IF SUPER^.Step(882, TRUE, 'Step number 882') THEN
    SUPER^.StepCompleteWhen((_runOneStep OR _runAllSteps) AND _finishStep);

    IF _runOneStep THEN
        _runOneStep := FALSE;
        RETURN;
    END_IF
END_IF

IF SUPER^.Step(883, TRUE, 'Step number 883') THEN
    SUPER^.StepCompleteWhen((_runOneStep OR _runAllSteps) AND _finishStep);

    IF _runOneStep THEN
        _runOneStep := FALSE;
        RETURN;
    END_IF
END_IF

IF SUPER^.Step(884, TRUE, 'Step number 884') THEN
    SUPER^.StepCompleteWhen((_runOneStep OR _runAllSteps) AND _finishStep);

    IF _runOneStep THEN
        _runOneStep := FALSE;
        RETURN;
    END_IF
END_IF

IF SUPER^.Step(885, TRUE, 'Step number 885') THEN
    SUPER^.StepCompleteWhen((_runOneStep OR _runAllSteps) AND _finishStep);

    IF _runOneStep THEN
        _runOneStep := FALSE;
        RETURN;
    END_IF
END_IF

IF SUPER^.Step(886, TRUE, 'Step number 886') THEN
    SUPER^.StepCompleteWhen((_runOneStep OR _runAllSteps) AND _finishStep);

    IF _runOneStep THEN
        _runOneStep := FALSE;
        RETURN;
    END_IF
END_IF

IF SUPER^.Step(887, TRUE, 'Step number 887') THEN
    SUPER^.StepCompleteWhen((_runOneStep OR _runAllSteps) AND _finishStep);

    IF _runOneStep THEN
        _runOneStep := FALSE;
        RETURN;
    END_IF
END_IF

IF SUPER^.Step(888, TRUE, 'Step number 888') THEN
    SUPER^.StepCompleteWhen((_runOneStep OR _runAllSteps) AND _finishStep);

    IF _runOneStep THEN
        _runOneStep := FALSE;
        RETURN;
    END_IF
END_IF

IF SUPER^.Step(889, TRUE, 'Step number 889') THEN
    SUPER^.StepCompleteWhen((_runOneStep OR _runAllSteps) AND _finishStep);

    IF _runOneStep THEN
        _runOneStep := FALSE;
        RETURN;
    END_IF
END_IF

IF SUPER^.Step(890, TRUE, 'Step number 890') THEN
    SUPER^.StepCompleteWhen((_runOneStep OR _runAllSteps) AND _finishStep);

    IF _runOneStep THEN
        _runOneStep := FALSE;
        RETURN;
    END_IF
END_IF

IF SUPER^.Step(891, TRUE, 'Step number 891') THEN
    SUPER^.StepCompleteWhen((_runOneStep OR _runAllSteps) AND _finishStep);

    IF _runOneStep THEN
        _runOneStep := FALSE;
        RETURN;
    END_IF
END_IF

IF SUPER^.Step(892, TRUE, 'Step number 892') THEN
    SUPER^.StepCompleteWhen((_runOneStep OR _runAllSteps) AND _finishStep);

    IF _runOneStep THEN
        _runOneStep := FALSE;
        RETURN;
    END_IF
END_IF

IF SUPER^.Step(893, TRUE, 'Step number 893') THEN
    SUPER^.StepCompleteWhen((_runOneStep OR _runAllSteps) AND _finishStep);

    IF _runOneStep THEN
        _runOneStep := FALSE;
        RETURN;
    END_IF
END_IF

IF SUPER^.Step(894, TRUE, 'Step number 894') THEN
    SUPER^.StepCompleteWhen((_runOneStep OR _runAllSteps) AND _finishStep);

    IF _runOneStep THEN
        _runOneStep := FALSE;
        RETURN;
    END_IF
END_IF

IF SUPER^.Step(895, TRUE, 'Step number 895') THEN
    SUPER^.StepCompleteWhen((_runOneStep OR _runAllSteps) AND _finishStep);

    IF _runOneStep THEN
        _runOneStep := FALSE;
        RETURN;
    END_IF
END_IF

IF SUPER^.Step(896, TRUE, 'Step number 896') THEN
    SUPER^.StepCompleteWhen((_runOneStep OR _runAllSteps) AND _finishStep);

    IF _runOneStep THEN
        _runOneStep := FALSE;
        RETURN;
    END_IF
END_IF

IF SUPER^.Step(897, TRUE, 'Step number 897') THEN
    SUPER^.StepCompleteWhen((_runOneStep OR _runAllSteps) AND _finishStep);

    IF _runOneStep THEN
        _runOneStep := FALSE;
        RETURN;
    END_IF
END_IF

IF SUPER^.Step(898, TRUE, 'Step number 898') THEN
    SUPER^.StepCompleteWhen((_runOneStep OR _runAllSteps) AND _finishStep);

    IF _runOneStep THEN
        _runOneStep := FALSE;
        RETURN;
    END_IF
END_IF

IF SUPER^.Step(899, TRUE, 'Step number 899') THEN
    SUPER^.StepCompleteWhen((_runOneStep OR _runAllSteps) AND _finishStep);

    IF _runOneStep THEN
        _runOneStep := FALSE;
        RETURN;
    END_IF
END_IF

IF SUPER^.Step(900, TRUE, 'Step number 900') THEN
    SUPER^.StepCompleteWhen((_runOneStep OR _runAllSteps) AND _finishStep);

    IF _runOneStep THEN
        _runOneStep := FALSE;
        RETURN;
    END_IF
END_IF

IF SUPER^.Step(901, TRUE, 'Step number 901') THEN
    SUPER^.StepCompleteWhen((_runOneStep OR _runAllSteps) AND _finishStep);

    IF _runOneStep THEN
        _runOneStep := FALSE;
        RETURN;
    END_IF
END_IF

IF SUPER^.Step(902, TRUE, 'Step number 902') THEN
    SUPER^.StepCompleteWhen((_runOneStep OR _runAllSteps) AND _finishStep);

    IF _runOneStep THEN
        _runOneStep := FALSE;
        RETURN;
    END_IF
END_IF

IF SUPER^.Step(903, TRUE, 'Step number 903') THEN
    SUPER^.StepCompleteWhen((_runOneStep OR _runAllSteps) AND _finishStep);

    IF _runOneStep THEN
        _runOneStep := FALSE;
        RETURN;
    END_IF
END_IF

IF SUPER^.Step(904, TRUE, 'Step number 904') THEN
    SUPER^.StepCompleteWhen((_runOneStep OR _runAllSteps) AND _finishStep);

    IF _runOneStep THEN
        _runOneStep := FALSE;
        RETURN;
    END_IF
END_IF

IF SUPER^.Step(905, TRUE, 'Step number 905') THEN
    SUPER^.StepCompleteWhen((_runOneStep OR _runAllSteps) AND _finishStep);

    IF _runOneStep THEN
        _runOneStep := FALSE;
        RETURN;
    END_IF
END_IF

IF SUPER^.Step(906, TRUE, 'Step number 906') THEN
    SUPER^.StepCompleteWhen((_runOneStep OR _runAllSteps) AND _finishStep);

    IF _runOneStep THEN
        _runOneStep := FALSE;
        RETURN;
    END_IF
END_IF

IF SUPER^.Step(907, TRUE, 'Step number 907') THEN
    SUPER^.StepCompleteWhen((_runOneStep OR _runAllSteps) AND _finishStep);

    IF _runOneStep THEN
        _runOneStep := FALSE;
        RETURN;
    END_IF
END_IF

IF SUPER^.Step(908, TRUE, 'Step number 908') THEN
    SUPER^.StepCompleteWhen((_runOneStep OR _runAllSteps) AND _finishStep);

    IF _runOneStep THEN
        _runOneStep := FALSE;
        RETURN;
    END_IF
END_IF

IF SUPER^.Step(909, TRUE, 'Step number 909') THEN
    SUPER^.StepCompleteWhen((_runOneStep OR _runAllSteps) AND _finishStep);

    IF _runOneStep THEN
        _runOneStep := FALSE;
        RETURN;
    END_IF
END_IF

IF SUPER^.Step(910, TRUE, 'Step number 910') THEN
    SUPER^.StepCompleteWhen((_runOneStep OR _runAllSteps) AND _finishStep);

    IF _runOneStep THEN
        _runOneStep := FALSE;
        RETURN;
    END_IF
END_IF

IF SUPER^.Step(911, TRUE, 'Step number 911') THEN
    SUPER^.StepCompleteWhen((_runOneStep OR _runAllSteps) AND _finishStep);

    IF _runOneStep THEN
        _runOneStep := FALSE;
        RETURN;
    END_IF
END_IF

IF SUPER^.Step(912, TRUE, 'Step number 912') THEN
    SUPER^.StepCompleteWhen((_runOneStep OR _runAllSteps) AND _finishStep);

    IF _runOneStep THEN
        _runOneStep := FALSE;
        RETURN;
    END_IF
END_IF

IF SUPER^.Step(913, TRUE, 'Step number 913') THEN
    SUPER^.StepCompleteWhen((_runOneStep OR _runAllSteps) AND _finishStep);

    IF _runOneStep THEN
        _runOneStep := FALSE;
        RETURN;
    END_IF
END_IF

IF SUPER^.Step(914, TRUE, 'Step number 914') THEN
    SUPER^.StepCompleteWhen((_runOneStep OR _runAllSteps) AND _finishStep);

    IF _runOneStep THEN
        _runOneStep := FALSE;
        RETURN;
    END_IF
END_IF

IF SUPER^.Step(915, TRUE, 'Step number 915') THEN
    SUPER^.StepCompleteWhen((_runOneStep OR _runAllSteps) AND _finishStep);

    IF _runOneStep THEN
        _runOneStep := FALSE;
        RETURN;
    END_IF
END_IF

IF SUPER^.Step(916, TRUE, 'Step number 916') THEN
    SUPER^.StepCompleteWhen((_runOneStep OR _runAllSteps) AND _finishStep);

    IF _runOneStep THEN
        _runOneStep := FALSE;
        RETURN;
    END_IF
END_IF

IF SUPER^.Step(917, TRUE, 'Step number 917') THEN
    SUPER^.StepCompleteWhen((_runOneStep OR _runAllSteps) AND _finishStep);

    IF _runOneStep THEN
        _runOneStep := FALSE;
        RETURN;
    END_IF
END_IF

IF SUPER^.Step(918, TRUE, 'Step number 918') THEN
    SUPER^.StepCompleteWhen((_runOneStep OR _runAllSteps) AND _finishStep);

    IF _runOneStep THEN
        _runOneStep := FALSE;
        RETURN;
    END_IF
END_IF

IF SUPER^.Step(919, TRUE, 'Step number 919') THEN
    SUPER^.StepCompleteWhen((_runOneStep OR _runAllSteps) AND _finishStep);

    IF _runOneStep THEN
        _runOneStep := FALSE;
        RETURN;
    END_IF
END_IF

IF SUPER^.Step(920, TRUE, 'Step number 920') THEN
    SUPER^.StepCompleteWhen((_runOneStep OR _runAllSteps) AND _finishStep);

    IF _runOneStep THEN
        _runOneStep := FALSE;
        RETURN;
    END_IF
END_IF

IF SUPER^.Step(921, TRUE, 'Step number 921') THEN
    SUPER^.StepCompleteWhen((_runOneStep OR _runAllSteps) AND _finishStep);

    IF _runOneStep THEN
        _runOneStep := FALSE;
        RETURN;
    END_IF
END_IF

IF SUPER^.Step(922, TRUE, 'Step number 922') THEN
    SUPER^.StepCompleteWhen((_runOneStep OR _runAllSteps) AND _finishStep);

    IF _runOneStep THEN
        _runOneStep := FALSE;
        RETURN;
    END_IF
END_IF

IF SUPER^.Step(923, TRUE, 'Step number 923') THEN
    SUPER^.StepCompleteWhen((_runOneStep OR _runAllSteps) AND _finishStep);

    IF _runOneStep THEN
        _runOneStep := FALSE;
        RETURN;
    END_IF
END_IF

IF SUPER^.Step(924, TRUE, 'Step number 924') THEN
    SUPER^.StepCompleteWhen((_runOneStep OR _runAllSteps) AND _finishStep);

    IF _runOneStep THEN
        _runOneStep := FALSE;
        RETURN;
    END_IF
END_IF

IF SUPER^.Step(925, TRUE, 'Step number 925') THEN
    SUPER^.StepCompleteWhen((_runOneStep OR _runAllSteps) AND _finishStep);

    IF _runOneStep THEN
        _runOneStep := FALSE;
        RETURN;
    END_IF
END_IF

IF SUPER^.Step(926, TRUE, 'Step number 926') THEN
    SUPER^.StepCompleteWhen((_runOneStep OR _runAllSteps) AND _finishStep);

    IF _runOneStep THEN
        _runOneStep := FALSE;
        RETURN;
    END_IF
END_IF

IF SUPER^.Step(927, TRUE, 'Step number 927') THEN
    SUPER^.StepCompleteWhen((_runOneStep OR _runAllSteps) AND _finishStep);

    IF _runOneStep THEN
        _runOneStep := FALSE;
        RETURN;
    END_IF
END_IF

IF SUPER^.Step(928, TRUE, 'Step number 928') THEN
    SUPER^.StepCompleteWhen((_runOneStep OR _runAllSteps) AND _finishStep);

    IF _runOneStep THEN
        _runOneStep := FALSE;
        RETURN;
    END_IF
END_IF

IF SUPER^.Step(929, TRUE, 'Step number 929') THEN
    SUPER^.StepCompleteWhen((_runOneStep OR _runAllSteps) AND _finishStep);

    IF _runOneStep THEN
        _runOneStep := FALSE;
        RETURN;
    END_IF
END_IF

IF SUPER^.Step(930, TRUE, 'Step number 930') THEN
    SUPER^.StepCompleteWhen((_runOneStep OR _runAllSteps) AND _finishStep);

    IF _runOneStep THEN
        _runOneStep := FALSE;
        RETURN;
    END_IF
END_IF

IF SUPER^.Step(931, TRUE, 'Step number 931') THEN
    SUPER^.StepCompleteWhen((_runOneStep OR _runAllSteps) AND _finishStep);

    IF _runOneStep THEN
        _runOneStep := FALSE;
        RETURN;
    END_IF
END_IF

IF SUPER^.Step(932, TRUE, 'Step number 932') THEN
    SUPER^.StepCompleteWhen((_runOneStep OR _runAllSteps) AND _finishStep);

    IF _runOneStep THEN
        _runOneStep := FALSE;
        RETURN;
    END_IF
END_IF

IF SUPER^.Step(933, TRUE, 'Step number 933') THEN
    SUPER^.StepCompleteWhen((_runOneStep OR _runAllSteps) AND _finishStep);

    IF _runOneStep THEN
        _runOneStep := FALSE;
        RETURN;
    END_IF
END_IF

IF SUPER^.Step(934, TRUE, 'Step number 934') THEN
    SUPER^.StepCompleteWhen((_runOneStep OR _runAllSteps) AND _finishStep);

    IF _runOneStep THEN
        _runOneStep := FALSE;
        RETURN;
    END_IF
END_IF

IF SUPER^.Step(935, TRUE, 'Step number 935') THEN
    SUPER^.StepCompleteWhen((_runOneStep OR _runAllSteps) AND _finishStep);

    IF _runOneStep THEN
        _runOneStep := FALSE;
        RETURN;
    END_IF
END_IF

IF SUPER^.Step(936, TRUE, 'Step number 936') THEN
    SUPER^.StepCompleteWhen((_runOneStep OR _runAllSteps) AND _finishStep);

    IF _runOneStep THEN
        _runOneStep := FALSE;
        RETURN;
    END_IF
END_IF

IF SUPER^.Step(937, TRUE, 'Step number 937') THEN
    SUPER^.StepCompleteWhen((_runOneStep OR _runAllSteps) AND _finishStep);

    IF _runOneStep THEN
        _runOneStep := FALSE;
        RETURN;
    END_IF
END_IF

IF SUPER^.Step(938, TRUE, 'Step number 938') THEN
    SUPER^.StepCompleteWhen((_runOneStep OR _runAllSteps) AND _finishStep);

    IF _runOneStep THEN
        _runOneStep := FALSE;
        RETURN;
    END_IF
END_IF

IF SUPER^.Step(939, TRUE, 'Step number 939') THEN
    SUPER^.StepCompleteWhen((_runOneStep OR _runAllSteps) AND _finishStep);

    IF _runOneStep THEN
        _runOneStep := FALSE;
        RETURN;
    END_IF
END_IF

IF SUPER^.Step(940, TRUE, 'Step number 940') THEN
    SUPER^.StepCompleteWhen((_runOneStep OR _runAllSteps) AND _finishStep);

    IF _runOneStep THEN
        _runOneStep := FALSE;
        RETURN;
    END_IF
END_IF

IF SUPER^.Step(941, TRUE, 'Step number 941') THEN
    SUPER^.StepCompleteWhen((_runOneStep OR _runAllSteps) AND _finishStep);

    IF _runOneStep THEN
        _runOneStep := FALSE;
        RETURN;
    END_IF
END_IF

IF SUPER^.Step(942, TRUE, 'Step number 942') THEN
    SUPER^.StepCompleteWhen((_runOneStep OR _runAllSteps) AND _finishStep);

    IF _runOneStep THEN
        _runOneStep := FALSE;
        RETURN;
    END_IF
END_IF

IF SUPER^.Step(943, TRUE, 'Step number 943') THEN
    SUPER^.StepCompleteWhen((_runOneStep OR _runAllSteps) AND _finishStep);

    IF _runOneStep THEN
        _runOneStep := FALSE;
        RETURN;
    END_IF
END_IF

IF SUPER^.Step(944, TRUE, 'Step number 944') THEN
    SUPER^.StepCompleteWhen((_runOneStep OR _runAllSteps) AND _finishStep);

    IF _runOneStep THEN
        _runOneStep := FALSE;
        RETURN;
    END_IF
END_IF

IF SUPER^.Step(945, TRUE, 'Step number 945') THEN
    SUPER^.StepCompleteWhen((_runOneStep OR _runAllSteps) AND _finishStep);

    IF _runOneStep THEN
        _runOneStep := FALSE;
        RETURN;
    END_IF
END_IF

IF SUPER^.Step(946, TRUE, 'Step number 946') THEN
    SUPER^.StepCompleteWhen((_runOneStep OR _runAllSteps) AND _finishStep);

    IF _runOneStep THEN
        _runOneStep := FALSE;
        RETURN;
    END_IF
END_IF

IF SUPER^.Step(947, TRUE, 'Step number 947') THEN
    SUPER^.StepCompleteWhen((_runOneStep OR _runAllSteps) AND _finishStep);

    IF _runOneStep THEN
        _runOneStep := FALSE;
        RETURN;
    END_IF
END_IF

IF SUPER^.Step(948, TRUE, 'Step number 948') THEN
    SUPER^.StepCompleteWhen((_runOneStep OR _runAllSteps) AND _finishStep);

    IF _runOneStep THEN
        _runOneStep := FALSE;
        RETURN;
    END_IF
END_IF

IF SUPER^.Step(949, TRUE, 'Step number 949') THEN
    SUPER^.StepCompleteWhen((_runOneStep OR _runAllSteps) AND _finishStep);

    IF _runOneStep THEN
        _runOneStep := FALSE;
        RETURN;
    END_IF
END_IF

IF SUPER^.Step(950, TRUE, 'Step number 950') THEN
    SUPER^.StepCompleteWhen((_runOneStep OR _runAllSteps) AND _finishStep);

    IF _runOneStep THEN
        _runOneStep := FALSE;
        RETURN;
    END_IF
END_IF

IF SUPER^.Step(951, TRUE, 'Step number 951') THEN
    SUPER^.StepCompleteWhen((_runOneStep OR _runAllSteps) AND _finishStep);

    IF _runOneStep THEN
        _runOneStep := FALSE;
        RETURN;
    END_IF
END_IF

IF SUPER^.Step(952, TRUE, 'Step number 952') THEN
    SUPER^.StepCompleteWhen((_runOneStep OR _runAllSteps) AND _finishStep);

    IF _runOneStep THEN
        _runOneStep := FALSE;
        RETURN;
    END_IF
END_IF

IF SUPER^.Step(953, TRUE, 'Step number 953') THEN
    SUPER^.StepCompleteWhen((_runOneStep OR _runAllSteps) AND _finishStep);

    IF _runOneStep THEN
        _runOneStep := FALSE;
        RETURN;
    END_IF
END_IF

IF SUPER^.Step(954, TRUE, 'Step number 954') THEN
    SUPER^.StepCompleteWhen((_runOneStep OR _runAllSteps) AND _finishStep);

    IF _runOneStep THEN
        _runOneStep := FALSE;
        RETURN;
    END_IF
END_IF

IF SUPER^.Step(955, TRUE, 'Step number 955') THEN
    SUPER^.StepCompleteWhen((_runOneStep OR _runAllSteps) AND _finishStep);

    IF _runOneStep THEN
        _runOneStep := FALSE;
        RETURN;
    END_IF
END_IF

IF SUPER^.Step(956, TRUE, 'Step number 956') THEN
    SUPER^.StepCompleteWhen((_runOneStep OR _runAllSteps) AND _finishStep);

    IF _runOneStep THEN
        _runOneStep := FALSE;
        RETURN;
    END_IF
END_IF

IF SUPER^.Step(957, TRUE, 'Step number 957') THEN
    SUPER^.StepCompleteWhen((_runOneStep OR _runAllSteps) AND _finishStep);

    IF _runOneStep THEN
        _runOneStep := FALSE;
        RETURN;
    END_IF
END_IF

IF SUPER^.Step(958, TRUE, 'Step number 958') THEN
    SUPER^.StepCompleteWhen((_runOneStep OR _runAllSteps) AND _finishStep);

    IF _runOneStep THEN
        _runOneStep := FALSE;
        RETURN;
    END_IF
END_IF

IF SUPER^.Step(959, TRUE, 'Step number 959') THEN
    SUPER^.StepCompleteWhen((_runOneStep OR _runAllSteps) AND _finishStep);

    IF _runOneStep THEN
        _runOneStep := FALSE;
        RETURN;
    END_IF
END_IF

IF SUPER^.Step(960, TRUE, 'Step number 960') THEN
    SUPER^.StepCompleteWhen((_runOneStep OR _runAllSteps) AND _finishStep);

    IF _runOneStep THEN
        _runOneStep := FALSE;
        RETURN;
    END_IF
END_IF

IF SUPER^.Step(961, TRUE, 'Step number 961') THEN
    SUPER^.StepCompleteWhen((_runOneStep OR _runAllSteps) AND _finishStep);

    IF _runOneStep THEN
        _runOneStep := FALSE;
        RETURN;
    END_IF
END_IF

IF SUPER^.Step(962, TRUE, 'Step number 962') THEN
    SUPER^.StepCompleteWhen((_runOneStep OR _runAllSteps) AND _finishStep);

    IF _runOneStep THEN
        _runOneStep := FALSE;
        RETURN;
    END_IF
END_IF

IF SUPER^.Step(963, TRUE, 'Step number 963') THEN
    SUPER^.StepCompleteWhen((_runOneStep OR _runAllSteps) AND _finishStep);

    IF _runOneStep THEN
        _runOneStep := FALSE;
        RETURN;
    END_IF
END_IF

IF SUPER^.Step(964, TRUE, 'Step number 964') THEN
    SUPER^.StepCompleteWhen((_runOneStep OR _runAllSteps) AND _finishStep);

    IF _runOneStep THEN
        _runOneStep := FALSE;
        RETURN;
    END_IF
END_IF

IF SUPER^.Step(965, TRUE, 'Step number 965') THEN
    SUPER^.StepCompleteWhen((_runOneStep OR _runAllSteps) AND _finishStep);

    IF _runOneStep THEN
        _runOneStep := FALSE;
        RETURN;
    END_IF
END_IF

IF SUPER^.Step(966, TRUE, 'Step number 966') THEN
    SUPER^.StepCompleteWhen((_runOneStep OR _runAllSteps) AND _finishStep);

    IF _runOneStep THEN
        _runOneStep := FALSE;
        RETURN;
    END_IF
END_IF

IF SUPER^.Step(967, TRUE, 'Step number 967') THEN
    SUPER^.StepCompleteWhen((_runOneStep OR _runAllSteps) AND _finishStep);

    IF _runOneStep THEN
        _runOneStep := FALSE;
        RETURN;
    END_IF
END_IF

IF SUPER^.Step(968, TRUE, 'Step number 968') THEN
    SUPER^.StepCompleteWhen((_runOneStep OR _runAllSteps) AND _finishStep);

    IF _runOneStep THEN
        _runOneStep := FALSE;
        RETURN;
    END_IF
END_IF

IF SUPER^.Step(969, TRUE, 'Step number 969') THEN
    SUPER^.StepCompleteWhen((_runOneStep OR _runAllSteps) AND _finishStep);

    IF _runOneStep THEN
        _runOneStep := FALSE;
        RETURN;
    END_IF
END_IF

IF SUPER^.Step(970, TRUE, 'Step number 970') THEN
    SUPER^.StepCompleteWhen((_runOneStep OR _runAllSteps) AND _finishStep);

    IF _runOneStep THEN
        _runOneStep := FALSE;
        RETURN;
    END_IF
END_IF

IF SUPER^.Step(971, TRUE, 'Step number 971') THEN
    SUPER^.StepCompleteWhen((_runOneStep OR _runAllSteps) AND _finishStep);

    IF _runOneStep THEN
        _runOneStep := FALSE;
        RETURN;
    END_IF
END_IF

IF SUPER^.Step(972, TRUE, 'Step number 972') THEN
    SUPER^.StepCompleteWhen((_runOneStep OR _runAllSteps) AND _finishStep);

    IF _runOneStep THEN
        _runOneStep := FALSE;
        RETURN;
    END_IF
END_IF

IF SUPER^.Step(973, TRUE, 'Step number 973') THEN
    SUPER^.StepCompleteWhen((_runOneStep OR _runAllSteps) AND _finishStep);

    IF _runOneStep THEN
        _runOneStep := FALSE;
        RETURN;
    END_IF
END_IF

IF SUPER^.Step(974, TRUE, 'Step number 974') THEN
    SUPER^.StepCompleteWhen((_runOneStep OR _runAllSteps) AND _finishStep);

    IF _runOneStep THEN
        _runOneStep := FALSE;
        RETURN;
    END_IF
END_IF

IF SUPER^.Step(975, TRUE, 'Step number 975') THEN
    SUPER^.StepCompleteWhen((_runOneStep OR _runAllSteps) AND _finishStep);

    IF _runOneStep THEN
        _runOneStep := FALSE;
        RETURN;
    END_IF
END_IF

IF SUPER^.Step(976, TRUE, 'Step number 976') THEN
    SUPER^.StepCompleteWhen((_runOneStep OR _runAllSteps) AND _finishStep);

    IF _runOneStep THEN
        _runOneStep := FALSE;
        RETURN;
    END_IF
END_IF

IF SUPER^.Step(977, TRUE, 'Step number 977') THEN
    SUPER^.StepCompleteWhen((_runOneStep OR _runAllSteps) AND _finishStep);

    IF _runOneStep THEN
        _runOneStep := FALSE;
        RETURN;
    END_IF
END_IF

IF SUPER^.Step(978, TRUE, 'Step number 978') THEN
    SUPER^.StepCompleteWhen((_runOneStep OR _runAllSteps) AND _finishStep);

    IF _runOneStep THEN
        _runOneStep := FALSE;
        RETURN;
    END_IF
END_IF

IF SUPER^.Step(979, TRUE, 'Step number 979') THEN
    SUPER^.StepCompleteWhen((_runOneStep OR _runAllSteps) AND _finishStep);

    IF _runOneStep THEN
        _runOneStep := FALSE;
        RETURN;
    END_IF
END_IF

IF SUPER^.Step(980, TRUE, 'Step number 980') THEN
    SUPER^.StepCompleteWhen((_runOneStep OR _runAllSteps) AND _finishStep);

    IF _runOneStep THEN
        _runOneStep := FALSE;
        RETURN;
    END_IF
END_IF

IF SUPER^.Step(981, TRUE, 'Step number 981') THEN
    SUPER^.StepCompleteWhen((_runOneStep OR _runAllSteps) AND _finishStep);

    IF _runOneStep THEN
        _runOneStep := FALSE;
        RETURN;
    END_IF
END_IF

IF SUPER^.Step(982, TRUE, 'Step number 982') THEN
    SUPER^.StepCompleteWhen((_runOneStep OR _runAllSteps) AND _finishStep);

    IF _runOneStep THEN
        _runOneStep := FALSE;
        RETURN;
    END_IF
END_IF

IF SUPER^.Step(983, TRUE, 'Step number 983') THEN
    SUPER^.StepCompleteWhen((_runOneStep OR _runAllSteps) AND _finishStep);

    IF _runOneStep THEN
        _runOneStep := FALSE;
        RETURN;
    END_IF
END_IF

IF SUPER^.Step(984, TRUE, 'Step number 984') THEN
    SUPER^.StepCompleteWhen((_runOneStep OR _runAllSteps) AND _finishStep);

    IF _runOneStep THEN
        _runOneStep := FALSE;
        RETURN;
    END_IF
END_IF

IF SUPER^.Step(985, TRUE, 'Step number 985') THEN
    SUPER^.StepCompleteWhen((_runOneStep OR _runAllSteps) AND _finishStep);

    IF _runOneStep THEN
        _runOneStep := FALSE;
        RETURN;
    END_IF
END_IF

IF SUPER^.Step(986, TRUE, 'Step number 986') THEN
    SUPER^.StepCompleteWhen((_runOneStep OR _runAllSteps) AND _finishStep);

    IF _runOneStep THEN
        _runOneStep := FALSE;
        RETURN;
    END_IF
END_IF

IF SUPER^.Step(987, TRUE, 'Step number 987') THEN
    SUPER^.StepCompleteWhen((_runOneStep OR _runAllSteps) AND _finishStep);

    IF _runOneStep THEN
        _runOneStep := FALSE;
        RETURN;
    END_IF
END_IF

IF SUPER^.Step(988, TRUE, 'Step number 988') THEN
    SUPER^.StepCompleteWhen((_runOneStep OR _runAllSteps) AND _finishStep);

    IF _runOneStep THEN
        _runOneStep := FALSE;
        RETURN;
    END_IF
END_IF

IF SUPER^.Step(989, TRUE, 'Step number 989') THEN
    SUPER^.StepCompleteWhen((_runOneStep OR _runAllSteps) AND _finishStep);

    IF _runOneStep THEN
        _runOneStep := FALSE;
        RETURN;
    END_IF
END_IF

IF SUPER^.Step(990, TRUE, 'Step number 990') THEN
    SUPER^.StepCompleteWhen((_runOneStep OR _runAllSteps) AND _finishStep);

    IF _runOneStep THEN
        _runOneStep := FALSE;
        RETURN;
    END_IF
END_IF

IF SUPER^.Step(991, TRUE, 'Step number 991') THEN
    SUPER^.StepCompleteWhen((_runOneStep OR _runAllSteps) AND _finishStep);

    IF _runOneStep THEN
        _runOneStep := FALSE;
        RETURN;
    END_IF
END_IF

IF SUPER^.Step(992, TRUE, 'Step number 992') THEN
    SUPER^.StepCompleteWhen((_runOneStep OR _runAllSteps) AND _finishStep);

    IF _runOneStep THEN
        _runOneStep := FALSE;
        RETURN;
    END_IF
END_IF

IF SUPER^.Step(993, TRUE, 'Step number 993') THEN
    SUPER^.StepCompleteWhen((_runOneStep OR _runAllSteps) AND _finishStep);

    IF _runOneStep THEN
        _runOneStep := FALSE;
        RETURN;
    END_IF
END_IF

IF SUPER^.Step(994, TRUE, 'Step number 994') THEN
    SUPER^.StepCompleteWhen((_runOneStep OR _runAllSteps) AND _finishStep);

    IF _runOneStep THEN
        _runOneStep := FALSE;
        RETURN;
    END_IF
END_IF

IF SUPER^.Step(995, TRUE, 'Step number 995') THEN
    SUPER^.StepCompleteWhen((_runOneStep OR _runAllSteps) AND _finishStep);

    IF _runOneStep THEN
        _runOneStep := FALSE;
        RETURN;
    END_IF
END_IF

IF SUPER^.Step(996, TRUE, 'Step number 996') THEN
    SUPER^.StepCompleteWhen((_runOneStep OR _runAllSteps) AND _finishStep);

    IF _runOneStep THEN
        _runOneStep := FALSE;
        RETURN;
    END_IF
END_IF

IF SUPER^.Step(997, TRUE, 'Step number 997') THEN
    SUPER^.StepCompleteWhen((_runOneStep OR _runAllSteps) AND _finishStep);

    IF _runOneStep THEN
        _runOneStep := FALSE;
        RETURN;
    END_IF
END_IF

IF SUPER^.Step(998, TRUE, 'Step number 998') THEN
    SUPER^.StepCompleteWhen((_runOneStep OR _runAllSteps) AND _finishStep);

    IF _runOneStep THEN
        _runOneStep := FALSE;
        RETURN;
    END_IF
END_IF

IF SUPER^.Step(999, TRUE, 'Step number 999') THEN
    SUPER^.StepCompleteWhen((_runOneStep OR _runAllSteps) AND _finishStep);

    IF _runOneStep THEN
        _runOneStep := FALSE;
        RETURN;
    END_IF
END_IF

IF SUPER^.Step(1000, TRUE, 'Step number 1000') THEN
    SUPER^.StepCompleteWhen((_runOneStep OR _runAllSteps) AND _finishStep);

    IF _runOneStep THEN
        _runOneStep := FALSE;
        RETURN;
    END_IF
END_IF

IF SUPER^.Step(1001, TRUE, 'Step number 1001') THEN
    SUPER^.StepCompleteWhen((_runOneStep OR _runAllSteps) AND _finishStep);

    IF _runOneStep THEN
        _runOneStep := FALSE;
        RETURN;
    END_IF
END_IF

IF SUPER^.Step(1002, TRUE, 'Step number 1002') THEN
    SUPER^.StepCompleteWhen((_runOneStep OR _runAllSteps) AND _finishStep);

    IF _runOneStep THEN
        _runOneStep := FALSE;
        RETURN;
    END_IF
END_IF

IF SUPER^.Step(1003, TRUE, 'Step number 1003') THEN
    SUPER^.StepCompleteWhen((_runOneStep OR _runAllSteps) AND _finishStep);

    IF _runOneStep THEN
        _runOneStep := FALSE;
        RETURN;
    END_IF
END_IF

IF SUPER^.Step(1004, TRUE, 'Step number 1004') THEN
    SUPER^.StepCompleteWhen((_runOneStep OR _runAllSteps) AND _finishStep);

    IF _runOneStep THEN
        _runOneStep := FALSE;
        RETURN;
    END_IF
END_IF

IF SUPER^.Step(1005, TRUE, 'Step number 1005') THEN
    SUPER^.StepCompleteWhen((_runOneStep OR _runAllSteps) AND _finishStep);

    IF _runOneStep THEN
        _runOneStep := FALSE;
        RETURN;
    END_IF
END_IF

IF SUPER^.Step(1006, TRUE, 'Step number 1006') THEN
    SUPER^.StepCompleteWhen((_runOneStep OR _runAllSteps) AND _finishStep);

    IF _runOneStep THEN
        _runOneStep := FALSE;
        RETURN;
    END_IF
END_IF

IF SUPER^.Step(1007, TRUE, 'Step number 1007') THEN
    SUPER^.StepCompleteWhen((_runOneStep OR _runAllSteps) AND _finishStep);

    IF _runOneStep THEN
        _runOneStep := FALSE;
        RETURN;
    END_IF
END_IF

IF SUPER^.Step(1008, TRUE, 'Step number 1008') THEN
    SUPER^.StepCompleteWhen((_runOneStep OR _runAllSteps) AND _finishStep);

    IF _runOneStep THEN
        _runOneStep := FALSE;
        RETURN;
    END_IF
END_IF

IF SUPER^.Step(1009, TRUE, 'Step number 1009') THEN
    SUPER^.StepCompleteWhen((_runOneStep OR _runAllSteps) AND _finishStep);

    IF _runOneStep THEN
        _runOneStep := FALSE;
        RETURN;
    END_IF
END_IF

IF SUPER^.Step(1010, TRUE, 'Step number 1010') THEN
    SUPER^.StepCompleteWhen((_runOneStep OR _runAllSteps) AND _finishStep);

    IF _runOneStep THEN
        _runOneStep := FALSE;
        RETURN;
    END_IF
END_IF

IF SUPER^.Step(1011, TRUE, 'Step number 1011') THEN
    SUPER^.StepCompleteWhen((_runOneStep OR _runAllSteps) AND _finishStep);

    IF _runOneStep THEN
        _runOneStep := FALSE;
        RETURN;
    END_IF
END_IF

IF SUPER^.Step(1012, TRUE, 'Step number 1012') THEN
    SUPER^.StepCompleteWhen((_runOneStep OR _runAllSteps) AND _finishStep);

    IF _runOneStep THEN
        _runOneStep := FALSE;
        RETURN;
    END_IF
END_IF

IF SUPER^.Step(1013, TRUE, 'Step number 1013') THEN
    SUPER^.StepCompleteWhen((_runOneStep OR _runAllSteps) AND _finishStep);

    IF _runOneStep THEN
        _runOneStep := FALSE;
        RETURN;
    END_IF
END_IF

IF SUPER^.Step(1014, TRUE, 'Step number 1014') THEN
    SUPER^.StepCompleteWhen((_runOneStep OR _runAllSteps) AND _finishStep);

    IF _runOneStep THEN
        _runOneStep := FALSE;
        RETURN;
    END_IF
END_IF

IF SUPER^.Step(1015, TRUE, 'Step number 1015') THEN
    SUPER^.StepCompleteWhen((_runOneStep OR _runAllSteps) AND _finishStep);

    IF _runOneStep THEN
        _runOneStep := FALSE;
        RETURN;
    END_IF
END_IF

IF SUPER^.Step(1016, TRUE, 'Step number 1016') THEN
    SUPER^.StepCompleteWhen((_runOneStep OR _runAllSteps) AND _finishStep);

    IF _runOneStep THEN
        _runOneStep := FALSE;
        RETURN;
    END_IF
END_IF

IF SUPER^.Step(1017, TRUE, 'Step number 1017') THEN
    SUPER^.StepCompleteWhen((_runOneStep OR _runAllSteps) AND _finishStep);

    IF _runOneStep THEN
        _runOneStep := FALSE;
        RETURN;
    END_IF
END_IF

IF SUPER^.Step(1018, TRUE, 'Step number 1018') THEN
    SUPER^.StepCompleteWhen((_runOneStep OR _runAllSteps) AND _finishStep);

    IF _runOneStep THEN
        _runOneStep := FALSE;
        RETURN;
    END_IF
END_IF

IF SUPER^.Step(1019, TRUE, 'Step number 1019') THEN
    SUPER^.StepCompleteWhen((_runOneStep OR _runAllSteps) AND _finishStep);

    IF _runOneStep THEN
        _runOneStep := FALSE;
        RETURN;
    END_IF
END_IF

IF SUPER^.Step(1020, TRUE, 'Step number 1020') THEN
    SUPER^.StepCompleteWhen((_runOneStep OR _runAllSteps) AND _finishStep);

    IF _runOneStep THEN
        _runOneStep := FALSE;
        RETURN;
    END_IF
END_IF

IF SUPER^.Step(1021, TRUE, 'Step number 1021') THEN
    SUPER^.StepCompleteWhen((_runOneStep OR _runAllSteps) AND _finishStep);

    IF _runOneStep THEN
        _runOneStep := FALSE;
        RETURN;
    END_IF
END_IF

IF SUPER^.Step(1022, TRUE, 'Step number 1022') THEN
    SUPER^.StepCompleteWhen((_runOneStep OR _runAllSteps) AND _finishStep);

    IF _runOneStep THEN
        _runOneStep := FALSE;
        RETURN;
    END_IF
END_IF

IF SUPER^.Step(1023, TRUE, 'Step number 1023') THEN
    SUPER^.StepCompleteWhen((_runOneStep OR _runAllSteps) AND _finishStep);

    IF _runOneStep THEN
        _runOneStep := FALSE;
        RETURN;
    END_IF
END_IF

//******************************************************************
IF SUPER^.Step(_stepId, _enabled, _stepDescription) THEN
    SUPER^.StepCompleteWhen((_runOneStep OR _runAllSteps) AND _finishStep);

    IF _runOneStep THEN
        _runOneStep := FALSE;
        RETURN;
    END_IF
END_IF
END_METHOD

METHOD MAIN_CommentOutPartOfRunningSequencer 
VAR 
	i : INT;
END_VAR
IF _sequenceRun =1 THEN
	IF Step(0, TRUE, 'Step 0') THEN
	   StepCompleteWhen(TRUE);
	END_IF

	IF Step(1, TRUE, 'Step 1') THEN
	   StepCompleteWhen(TRUE);
	END_IF

	IF Step(2, TRUE, 'Step 2') THEN
	   StepCompleteWhen(TRUE);
	END_IF

	IF Step(3, TRUE, 'Step 3') THEN
			StepCompleteWhen(FALSE);
	END_IF
	
	FOR i := 4 TO _totalStepNumber-2 DO
		IF Step(i, TRUE, CONCAT('Step ', INT_TO_STRING(i))) THEN
			StepCompleteWhen(FALSE);
		END_IF
	END_FOR
	
	IF Step(_totalStepNumber - 1, TRUE, CONCAT('Step ', INT_TO_STRING(_totalStepNumber - 1))) THEN
	  _SequenceComplete();
	END_IF
END_IF

IF _sequenceRun >=2 THEN
	IF Step(0, TRUE, 'Step 0') THEN
	   StepCompleteWhen(TRUE);
	END_IF

//	IF Step(1, TRUE, 'Step 1') THEN
//	   StepCompleteWhen(TRUE);
//	END_IF

//	IF Step(2, TRUE, 'Step 2') THEN
//	   StepCompleteWhen(TRUE);
//	END_IF

	IF Step(3, TRUE, 'Step 3') THEN
	   StepCompleteWhen(FALSE);
	END_IF
	
	FOR i := 4 TO _totalStepNumber-2 DO
		IF Step(i, TRUE, CONCAT('Step ', INT_TO_STRING(i))) THEN
			StepCompleteWhen(FALSE);
		END_IF
	END_FOR
	
	IF Step(_totalStepNumber - 1, TRUE, CONCAT('Step ', INT_TO_STRING(_totalStepNumber - 1))) THEN
	  _SequenceComplete();
	END_IF
END_IF
END_METHOD

METHOD MAIN_ExecutionInOnePLCcycle 
VAR 
	i : INT;
END_VAR
FOR i := 0 TO _totalStepNumber-2 DO
    IF Step(i, TRUE, CONCAT('Step ', INT_TO_STRING(i))) THEN
        StepCompleteWhen(TRUE);
    END_IF
END_FOR

IF Step(_totalStepNumber - 1, TRUE, CONCAT('Step ', INT_TO_STRING(_totalStepNumber - 1))) THEN
   	_SequenceComplete();
END_IF
END_METHOD

METHOD MAIN_MaxStepId 
VAR 
	i : INT;
END_VAR
FOR i := 0 TO _totalStepNumber-1 DO
    IF Step(i, TRUE, CONCAT('Step ', INT_TO_STRING(i))) THEN
        StepCompleteWhen(_finishStep);
    END_IF
END_FOR
IF Step(_stepId, TRUE, CONCAT('Step ', INT_TO_STRING(_stepId))) THEN
    StepCompleteWhen(TRUE);
END_IF
END_METHOD

METHOD MAIN_MinStepId 
VAR 
	i : INT;
END_VAR
IF Step(_stepId, TRUE, CONCAT('Step ', INT_TO_STRING(_stepId))) THEN
    StepCompleteWhen(TRUE);
END_IF

FOR i := 1 TO _totalStepNumber-1 DO
    IF Step(i, TRUE, CONCAT('Step ', INT_TO_STRING(i))) THEN
        StepCompleteWhen(_finishStep);
    END_IF
END_FOR
END_METHOD

METHOD MAIN_NumberOfStepsCount 
VAR 
	i : INT;
END_VAR
IF Step(0, TRUE, 'Step 0') THEN
    StepCompleteWhen(TRUE);
END_IF

FOR i := 1 TO _totalStepNumber - 1 DO
    IF Step(i, TRUE, CONCAT('Step ', INT_TO_STRING(i))) THEN
        StepCompleteWhen(_finishStep);
    END_IF
END_FOR
END_METHOD

METHOD MAIN_OnStateChangeWhenChangingModes 
VAR 
	i : INT;
END_VAR
IF _sequenceRun <= _cyclicCycles OR _sequenceRun > _cyclicCycles + _stepInEvents + 1 THEN
    SetCyclicMode();

    FOR i := 0 TO _totalStepNumber - 2 DO
        IF Step(i, TRUE, CONCAT('Step ', INT_TO_STRING(i))) THEN
            _StepCompleteWhen(TRUE);
        END_IF
    END_FOR

    IF Step(_totalStepNumber - 1, TRUE, CONCAT('Step ', INT_TO_STRING(_totalStepNumber - 1))) THEN
        CompleteSequence();
		_sequenceCycles := _sequenceCycles + 1;
    END_IF
END_IF
IF _sequenceRun = _cyclicCycles+1 THEN
    SetStepMode();
	Step(0,FALSE,'');	
END_IF
IF _sequenceRun > _cyclicCycles+1  AND _sequenceRun <= _cyclicCycles + _stepInEvents +1 THEN
    SetStepMode();
	_StepIn();
    FOR i := 0 TO _totalStepNumber - 2 DO
        IF Step(i, TRUE, CONCAT('Step ', INT_TO_STRING(i))) THEN
            _StepCompleteWhen(TRUE);
        END_IF
    END_FOR

    IF Step(_totalStepNumber - 1, TRUE, CONCAT('Step ', INT_TO_STRING(_totalStepNumber - 1))) THEN
        CompleteSequence();
		_sequenceCycles := _sequenceCycles + 1;
    END_IF
END_IF
END_METHOD

METHOD MAIN_RequestStep 
VAR 
	i : INT;
END_VAR
IF _sequenceRun =1 THEN
	FOR i := -5 TO -1 DO
		IF Step(i, TRUE, CONCAT('Step ', INT_TO_STRING(i))) THEN
			StepCompleteWhen(TRUE);
		END_IF
	END_FOR
	
	IF Step(0, TRUE, 'Step 0') THEN
		RequestStep(-5);
	END_IF
	
	FOR i := 1 TO 5 DO
		IF Step(i, TRUE, CONCAT('Step ', INT_TO_STRING(i))) THEN
			StepCompleteWhen(TRUE);
		END_IF
	END_FOR
END_IF

IF _sequenceRun =2 THEN
	FOR i := -5 TO 5 DO
		IF Step(i, TRUE, CONCAT('Step ', INT_TO_STRING(i))) THEN
			StepCompleteWhen(FALSE);
		END_IF
	END_FOR
END_IF

IF _sequenceRun =3 THEN
	IF Step(-5, TRUE, 'Step -5') THEN
		RequestStep(0);
	END_IF

	FOR i := -4 TO 5 DO
		IF Step(i, TRUE, CONCAT('Step ', INT_TO_STRING(i))) THEN
			StepCompleteWhen(FALSE);
		END_IF
	END_FOR
END_IF
END_METHOD

METHOD MAIN_RequestStepFromHigherToLower 
VAR 
	i : INT;
END_VAR
IF _sequenceRun = 1 THEN
    FOR i := 0 TO _reqStep + 4 DO
        IF Step(i, TRUE, CONCAT('Step ', INT_TO_STRING(i))) THEN
            StepCompleteWhen(TRUE);
        END_IF
    END_FOR

    FOR i := _reqStep + 5 TO _totalStepNumber - 2 DO
        Step(i, TRUE, CONCAT('Step ', INT_TO_STRING(i)));
    END_FOR

    RequestStep(_reqStep);

    IF Step(_totalStepNumber - 1, TRUE, CONCAT('Step ', INT_TO_STRING(_totalStepNumber - 1))) THEN
        _SequenceComplete();
    END_IF
END_IF

IF _sequenceRun = 2 THEN
    FOR i := 0 TO _totalStepNumber - 2 DO
        Step(i, TRUE, CONCAT('Step ', INT_TO_STRING(i)));
    END_FOR

    IF Step(_totalStepNumber - 1, TRUE, CONCAT('Step ', INT_TO_STRING(_totalStepNumber - 1))) THEN
        _SequenceComplete();
    END_IF
END_IF
END_METHOD

METHOD MAIN_RequestStepFromLowerToHigher 
VAR 
	i : INT;
END_VAR
IF _sequenceRun = 1 THEN
    IF Step(0, TRUE, 'Step 0') THEN
        StepCompleteWhen(TRUE);
    END_IF

    FOR i := 1 TO _totalStepNumber - 2 DO
        Step(i, TRUE, CONCAT('Step ', INT_TO_STRING(i)));
    END_FOR

    IF Step(_totalStepNumber - 1, TRUE, CONCAT('Step ', INT_TO_STRING(_totalStepNumber - 1))) THEN
        _SequenceComplete();
    END_IF
END_IF

IF _sequenceRun = 2 THEN
    IF Step(0, TRUE, 'Step 0') THEN
        StepCompleteWhen(TRUE);
    END_IF

    RequestStep(_reqStep);

    FOR i := 1 TO _totalStepNumber - 2 DO
        Step(i, TRUE, CONCAT('Step ', INT_TO_STRING(i)));
    END_FOR

    IF Step(_totalStepNumber - 1, TRUE, CONCAT('Step ', INT_TO_STRING(_totalStepNumber - 1))) THEN
        _SequenceComplete();
    END_IF
END_IF
END_METHOD

METHOD MAIN_RequestStepToFirstStepWithStepId0 
VAR 
	i : INT;
END_VAR
FOR i := 0 TO 4 DO
    IF Step(i, TRUE, CONCAT('Step ', INT_TO_STRING(i))) THEN
        StepCompleteWhen(_finishStep);
    END_IF
END_FOR

IF Step(5, TRUE, 'Step 5') THEN
    RequestStep(0);
END_IF

FOR i := 6 TO _totalStepNumber DO
    IF Step(i, TRUE, CONCAT('Step ', INT_TO_STRING(i))) THEN
        StepCompleteWhen(_finishStep);
    END_IF
END_FOR
END_METHOD

METHOD MAIN_RequestStepToNotExistingStep 
VAR 
	i : INT;
END_VAR
IF _sequenceRun = 1 THEN
    RequestStep(_reqStepNotExists);

    FOR i := 0 TO _totalStepNumber - 2 DO
        Step(i, TRUE, CONCAT('Step ', INT_TO_STRING(i)));
    END_FOR

    IF Step(_totalStepNumber - 1, TRUE, CONCAT('Step ', INT_TO_STRING(_totalStepNumber - 1))) THEN
        _SequenceComplete();
    END_IF
END_IF

IF _sequenceRun >= 2 THEN
    FOR i := 0 TO _totalStepNumber - 2 DO
        Step(i, TRUE, CONCAT('Step ', INT_TO_STRING(i)));
    END_FOR

    IF Step(_totalStepNumber - 1, TRUE, CONCAT('Step ', INT_TO_STRING(_totalStepNumber - 1))) THEN
        _SequenceComplete();
    END_IF
END_IF
END_METHOD

METHOD MAIN_RequestStepWhilePreviousRequestStepHasNotBeenYetProcessed 
VAR 
	i : INT;
END_VAR
FOR i := 0 TO _reqStep + 4 DO
    IF Step(i, TRUE, CONCAT('Step ', INT_TO_STRING(i))) THEN
        StepCompleteWhen(TRUE);
    END_IF
END_FOR

RequestStep(_reqStep);

FOR i := _reqStep + 5 TO _totalStepNumber - 2 DO
    Step(i, TRUE, CONCAT('Step ', INT_TO_STRING(i)));
END_FOR

RequestStep(_reqStep + 10);

IF Step(_totalStepNumber - 1, TRUE, CONCAT('Step ', INT_TO_STRING(_totalStepNumber - 1))) THEN
    _SequenceComplete();
END_IF
END_METHOD

METHOD MAIN_RestoreChildBetweenSteps 
VAR 
	i : INT;
	_childState : INT;
END_VAR
FOR i := 0 TO _totalStepNumber-2 DO
    IF Step(i, TRUE, CONCAT('Step ', INT_TO_STRING(i))) THEN
		_childState := _myTcoChildState.State;
		_myTcoChildState.ChangeState(_myTcoChildState._requestedState);
        StepCompleteWhen(TRUE);
    END_IF
END_FOR

IF Step(_totalStepNumber - 1, TRUE, CONCAT('Step ', INT_TO_STRING(_totalStepNumber - 1))) THEN
   	_SequenceComplete();
END_IF
END_METHOD

METHOD MAIN_SetStepMode 
VAR 
	i : INT;
END_VAR
IF _sequenceRun = 1 THEN
    IF Step(0, TRUE, 'Initial step') THEN
        StepCompleteWhen(TRUE);
    END_IF

    FOR i := 1 TO _totalStepNumber - 2 DO
        Step(i, TRUE, CONCAT('Step ', INT_TO_STRING(i)));
    END_FOR

    IF Step(_totalStepNumber - 1, TRUE, CONCAT('Step ', INT_TO_STRING(_totalStepNumber - 1))) THEN
        _SequenceComplete();
    END_IF
END_IF

IF _sequenceRun =4 THEN
    IF Step(0, TRUE, 'Initial step') THEN
        StepCompleteWhen(TRUE);
    END_IF

    FOR i := 1 TO _totalStepNumber - 2 DO
        IF Step(i, TRUE, CONCAT('Step ', INT_TO_STRING(i))) THEN
	        StepCompleteWhen(TRUE);
		END_IF
    END_FOR

    IF Step(_totalStepNumber - 1, TRUE, CONCAT('Step ', INT_TO_STRING(_totalStepNumber - 1))) THEN
        _SequenceComplete();
    END_IF
END_IF
END_METHOD

METHOD MAIN_StepMode 
VAR 
	i : INT;
END_VAR
IF _sequenceRun = 1 THEN
    IF Step(0, TRUE, 'Initial step') THEN
        StepCompleteWhen(TRUE);
    END_IF

    FOR i := 1 TO _totalStepNumber - 2 DO
        Step(i, TRUE, CONCAT('Step ', INT_TO_STRING(i)));
    END_FOR

    IF Step(_totalStepNumber - 1, TRUE, CONCAT('Step ', INT_TO_STRING(_totalStepNumber - 1))) THEN
        _SequenceComplete();
    END_IF
END_IF

IF _sequenceRun > 1 THEN
    _StepIn();

    IF Step(0, TRUE, 'Initial step') THEN
        StepCompleteWhen(TRUE);
    END_IF

    FOR i := 1 TO _totalStepNumber - 2 DO
        IF Step(i, TRUE, CONCAT('Step ', INT_TO_STRING(i))) THEN
            StepCompleteWhen(TRUE);
        END_IF
    END_FOR

    IF Step(_totalStepNumber - 1, TRUE, CONCAT('Step ', INT_TO_STRING(_totalStepNumber - 1))) THEN
        _SequenceComplete();
    END_IF
END_IF
END_METHOD

METHOD MAIN_StepModeChangeStepIdDuringExecution 
VAR 
	i : INT;
END_VAR
IF _sequenceRun = 1 THEN
    IF _currentStep.Status = 20 THEN
       _StepIn();
    END_IF

    // Step 0
    IF Step(0, TRUE, 'Step 0') THEN
        StepCompleteWhen(TRUE);
    END_IF

    // Step 1
    IF Step(1, TRUE, 'Step 1') THEN
        StepCompleteWhen(TRUE);
    END_IF

    // Step 2
    IF Step(2, TRUE, 'Step 2') THEN
        StepCompleteWhen(TRUE);
    END_IF

    // Step 3
    IF Step(3, TRUE, 'Step 3') THEN
        StepCompleteWhen(FALSE);
    END_IF

    FOR i := 4 TO _totalStepNumber - 2 DO
        Step(i, TRUE, CONCAT('Step  ', INT_TO_STRING(i)));
    END_FOR

    IF Step(_totalStepNumber - 1, TRUE, CONCAT('Step  ', INT_TO_STRING(_totalStepNumber - 1))) THEN
        _SequenceComplete();
    END_IF
END_IF
IF _sequenceRun = 2 THEN
    IF _currentStep.Status = 20 THEN
       _StepIn();
    END_IF

    // Step 0
    IF Step(0, TRUE, 'Step 0') THEN
        StepCompleteWhen(TRUE);
    END_IF

    // Step 1
    IF Step(1, TRUE, 'Step 1') THEN
        StepCompleteWhen(TRUE);
    END_IF

    // Step 2
    IF Step(2, TRUE, 'Step 2') THEN
        StepCompleteWhen(TRUE);
    END_IF

    // Step 3
    IF Step(5, TRUE, 'Step 3') THEN
        StepCompleteWhen(FALSE);
    END_IF

    FOR i := 4 TO _totalStepNumber - 2 DO
        Step(i, TRUE, CONCAT('Step  ', INT_TO_STRING(i)));
    END_FOR

    IF Step(_totalStepNumber - 1, TRUE, CONCAT('Step  ', INT_TO_STRING(_totalStepNumber - 1))) THEN
        _SequenceComplete();
    END_IF
END_IF
END_METHOD

METHOD MAIN_StepModeChangeStepOrder 
VAR 
	i : INT;
END_VAR
IF _sequenceRun <= _totalStepNumber + 1 THEN
    IF _currentStep.Status = 20 THEN
       _StepIn();
    END_IF

    // Step 0
    IF Step(0, TRUE, 'Step 0') THEN
        StepCompleteWhen(TRUE);
    END_IF

    // Step 1
    IF Step(1, TRUE, 'Step 1') THEN
        StepCompleteWhen(TRUE);
    END_IF

    // Step 2
    IF Step(2, TRUE, 'Step 2') THEN
        StepCompleteWhen(TRUE);
    END_IF

    // Step 3
    IF Step(3, TRUE, 'Step 3') THEN
        StepCompleteWhen(FALSE);
    END_IF

    FOR i := 4 TO _totalStepNumber - 2 DO
        Step(i, TRUE, CONCAT('Step  ', INT_TO_STRING(i)));
    END_FOR

    IF Step(_totalStepNumber-1, TRUE, CONCAT('Step  ', INT_TO_STRING(_totalStepNumber-1))) THEN
        _SequenceComplete();
    END_IF
END_IF
IF _sequenceRun = _totalStepNumber + 2 THEN
    IF _currentStep.Status = 20 THEN
       _StepIn();
    END_IF

    // Step 0
    IF Step(0, TRUE, 'Step 0') THEN
        StepCompleteWhen(TRUE);
    END_IF

    // Step 1
    IF Step(1, TRUE, 'Step 1') THEN
        StepCompleteWhen(TRUE);
    END_IF

    // Step 3
    IF Step(3, TRUE, 'Step 3') THEN
        StepCompleteWhen(FALSE);
    END_IF

    // Step 2
    IF Step(2, TRUE, 'Step 2') THEN
        StepCompleteWhen(TRUE);
    END_IF

    FOR i := 4 TO _totalStepNumber - 2 DO
        Step(i, TRUE, CONCAT('Step  ', INT_TO_STRING(i)));
    END_FOR

    IF Step(_totalStepNumber-1, TRUE, CONCAT('Step  ', INT_TO_STRING(_totalStepNumber-1))) THEN
        _SequenceComplete();
    END_IF
END_IF
END_METHOD

METHOD MAIN_StepModeCommentOutPartOfRunningSequencer 
VAR 
	i : INT;
END_VAR
IF _sequenceRun =1 THEN
    IF (_currentStep.Status = 20) THEN
        _StepIn();
    END_IF

	IF Step(0, TRUE, 'Step 0') THEN
	   StepCompleteWhen(TRUE);
	END_IF

	IF Step(1, TRUE, 'Step 1') THEN
	   StepCompleteWhen(TRUE);
	END_IF

	IF Step(2, TRUE, 'Step 2') THEN
	   StepCompleteWhen(TRUE);
	END_IF

	IF Step(3, TRUE, 'Step 3') THEN
			StepCompleteWhen(FALSE);
	END_IF
	
	FOR i := 4 TO _totalStepNumber-2 DO
		IF Step(i, TRUE, CONCAT('Step ', INT_TO_STRING(i))) THEN
			StepCompleteWhen(FALSE);
		END_IF
	END_FOR
	
	IF Step(_totalStepNumber-1, TRUE, CONCAT('Step ', INT_TO_STRING(_totalStepNumber-1))) THEN
	  _SequenceComplete();
	END_IF
END_IF

IF _sequenceRun >=2 THEN
    IF (_currentStep.Status = 20) THEN
        _StepIn();
    END_IF

	IF Step(0, TRUE, 'Step 0') THEN
	   StepCompleteWhen(TRUE);
	END_IF

//	IF Step(1, TRUE, 'Step 1') THEN
//	   StepCompleteWhen(TRUE);
//	END_IF

//	IF Step(2, TRUE, 'Step 2') THEN
//	   StepCompleteWhen(TRUE);
//	END_IF

	IF Step(3, TRUE, 'Step 3') THEN
	   StepCompleteWhen(FALSE);
	END_IF
	
	FOR i := 4 TO _totalStepNumber-2 DO
		IF Step(i, TRUE, CONCAT('Step ', INT_TO_STRING(i))) THEN
			StepCompleteWhen(FALSE);
		END_IF
	END_FOR
	
	IF Step(_totalStepNumber-1, TRUE, CONCAT('Step ', INT_TO_STRING(_totalStepNumber-1))) THEN
	  _SequenceComplete();
	END_IF
END_IF
END_METHOD

METHOD MAIN_StepModeDisabledStep 
VAR 
	i : INT;
END_VAR
IF _sequenceRun = 1 THEN
    FOR i := 0 TO _totalStepNumber-1 DO
        Step(i, TRUE, CONCAT('Step ', INT_TO_STRING(i)));
    END_FOR
END_IF

IF _sequenceRun = 2 OR _sequenceRun = 3 THEN
    IF _sequenceRun = 2 THEN
        _StepIn();
    END_IF

    IF Step(0, TRUE, 'Step 0') THEN
        StepCompleteWhen(TRUE);
    END_IF

    FOR i := 1 TO _totalStepNumber - 2 DO
        Step(i, TRUE, CONCAT('Step ', INT_TO_STRING(i)));
    END_FOR

    IF Step(_totalStepNumber-1, TRUE, CONCAT('Step ', INT_TO_STRING(_totalStepNumber-1))) THEN
        CompleteSequence();
    END_IF
END_IF

IF _sequenceRun = 4 THEN
    IF Step(0, TRUE, 'Step 0') THEN
        StepCompleteWhen(TRUE);
    END_IF

    IF Step(1, FALSE, 'Step 1') THEN
        StepCompleteWhen(TRUE);
    END_IF

    FOR i := 2 TO _totalStepNumber - 2 DO
        Step(i, TRUE, CONCAT('Step ', INT_TO_STRING(i)));
    END_FOR

    IF Step(_totalStepNumber-1, TRUE, CONCAT('Step ', INT_TO_STRING(_totalStepNumber-1))) THEN
        CompleteSequence();
    END_IF
END_IF

IF _sequenceRun >= 5 THEN
    _StepIn();

    IF Step(0, TRUE, 'Step 0') THEN
        StepCompleteWhen(TRUE);
    END_IF

    IF Step(1, FALSE, 'Step 1') THEN
        StepCompleteWhen(TRUE);
    END_IF

    FOR i := 2 TO _totalStepNumber - 2 DO
        Step(i, TRUE, CONCAT('Step ', INT_TO_STRING(i)));
    END_FOR

    IF Step(_totalStepNumber-1, TRUE, CONCAT('Step ', INT_TO_STRING(_totalStepNumber-1))) THEN
        CompleteSequence();
    END_IF
END_IF
END_METHOD

METHOD MAIN_StepModeRequestStepFromHigherToLower 
VAR 
	i : INT;
END_VAR
IF _sequenceRun <=_reqStep + 5 THEN
    FOR i := 0 TO _reqStep + 4 DO
       _StepIn();
        IF Step(i, TRUE, CONCAT('Step ', INT_TO_STRING(i))) THEN
            StepCompleteWhen(TRUE);
        END_IF
    END_FOR

    FOR i := _reqStep + 5 TO _totalStepNumber - 2 DO
       _StepIn();
        Step(i, TRUE, CONCAT('Step ', INT_TO_STRING(i)));
    END_FOR

    IF Step(_totalStepNumber-1, TRUE, CONCAT('Step ', INT_TO_STRING(_totalStepNumber-1))) THEN
        _SequenceComplete();
    END_IF
END_IF

IF _sequenceRun =_reqStep + 6 THEN
    FOR i := 0 TO _reqStep + 4 DO
       _StepIn();
        IF Step(i, TRUE, CONCAT('Step ', INT_TO_STRING(i))) THEN
            StepCompleteWhen(TRUE);
        END_IF
    END_FOR

    FOR i := _reqStep + 5 TO _totalStepNumber - 2 DO
       _StepIn();
        Step(i, TRUE, CONCAT('Step ', INT_TO_STRING(i)));
    END_FOR

    RequestStep(_reqStep);

    IF Step(_totalStepNumber-1, TRUE, CONCAT('Step ', INT_TO_STRING(_totalStepNumber-1))) THEN
        _SequenceComplete();
    END_IF
END_IF

IF _sequenceRun >=_reqStep + 7 THEN
    FOR i := 0 TO _totalStepNumber - 2 DO
       _StepIn();
        Step(i, TRUE, CONCAT('Step ', INT_TO_STRING(i)));
    END_FOR

    IF Step(_totalStepNumber-1, TRUE, CONCAT('Step ', INT_TO_STRING(_totalStepNumber-1))) THEN
        _SequenceComplete();
    END_IF
END_IF
END_METHOD

METHOD MAIN_StepModeRequestStepFromLowerToHigher 
VAR 
	i : INT;
END_VAR
IF _sequenceRun = 1 THEN
    IF _currentStep.Status = 20 THEN
       _StepIn();
    END_IF
    IF Step(0, TRUE, 'Step 0') THEN
        StepCompleteWhen(TRUE);
    END_IF

    FOR i := 1 TO _totalStepNumber - 2 DO
        Step(i, TRUE, CONCAT('Step ', INT_TO_STRING(i)));
    END_FOR

    IF Step(_totalStepNumber-1, TRUE, CONCAT('Step ', INT_TO_STRING(_totalStepNumber-1))) THEN
        _SequenceComplete();
    END_IF
END_IF

IF _sequenceRun = 2 THEN
    IF _currentStep.Status = 20 THEN
       _StepIn();
    END_IF
    IF Step(0, TRUE, 'Step 0') THEN
        StepCompleteWhen(TRUE);
    END_IF

    RequestStep(_reqStep);

    FOR i := 1 TO _totalStepNumber - 2 DO
        Step(i, TRUE, CONCAT('Step ', INT_TO_STRING(i)));
    END_FOR

    IF Step(_totalStepNumber-1, TRUE, CONCAT('Step ', INT_TO_STRING(_totalStepNumber-1))) THEN
        _SequenceComplete();
    END_IF
END_IF
END_METHOD

METHOD MAIN_StepModeStepBackwardFromRunningStep 
VAR 
	i : INT;
END_VAR
IF _sequenceRun = 1 THEN
    _StepIn();
END_IF

IF _sequenceRun = 11 THEN
    _StepBackward();
END_IF

Step(0, TRUE, 'Step 0');
Step(1, TRUE, 'Step 1');

IF Step(2, TRUE, 'Step 2') THEN
    _StepCompleteWhen(_sequenceRun >= 20);
END_IF

IF Step(3, TRUE, 'Step 3') THEN
    _StepCompleteWhen(_sequenceRun >= 20);
END_IF

FOR i := 4 TO _totalStepNumber - 2 DO
    Step(i, TRUE, CONCAT('Step ', INT_TO_STRING(i)));
END_FOR

IF Step(_totalStepNumber-1, TRUE, CONCAT('Step ', INT_TO_STRING(_totalStepNumber-1))) THEN
    CompleteSequence();
END_IF
END_METHOD

METHOD MAIN_StepModeStepForwardBackward 
VAR 
	i : INT;
END_VAR
IF _sequenceRun = 1 THEN
    FOR i := 0 TO _totalStepNumber - 2 DO
        Step(i, TRUE, CONCAT('Step ', INT_TO_STRING(i)));
    END_FOR

    IF Step(_totalStepNumber - 1, TRUE, CONCAT('Step ', INT_TO_STRING(_totalStepNumber - 1))) THEN
        CompleteSequence();
    END_IF
END_IF

IF _sequenceRun = 2 THEN
    _StepIn();

    IF Step(0, TRUE, 'Step 0') THEN
        StepCompleteWhen(TRUE);
    END_IF

    FOR i := 1 TO _totalStepNumber - 2 DO
        Step(i, TRUE, CONCAT('Step ', INT_TO_STRING(i)));
    END_FOR

    IF Step(_totalStepNumber - 1, TRUE, CONCAT('Step ', INT_TO_STRING(_totalStepNumber- 1))) THEN
        CompleteSequence();
    END_IF
END_IF

IF _sequenceRun = 3 OR _sequenceRun = 5 THEN
    _StepForward();

    IF Step(0, TRUE, 'Step 0') THEN
        StepCompleteWhen(TRUE);
    END_IF

    FOR i := 1 TO _totalStepNumber - 2 DO
        Step(i, TRUE, CONCAT('Step ', INT_TO_STRING(i)));
    END_FOR

    IF Step(_totalStepNumber - 1, TRUE, CONCAT('Step ', INT_TO_STRING(_totalStepNumber - 1))) THEN
        CompleteSequence();
    END_IF
END_IF

IF _sequenceRun = 4 THEN
    RequestStep(_totalStepNumber -1);

    IF Step(0, TRUE, 'Step 0') THEN
        StepCompleteWhen(TRUE);
    END_IF

    FOR i := 1 TO _totalStepNumber - 2 DO
        Step(i, TRUE, CONCAT('Step ', INT_TO_STRING(i)));
    END_FOR

    IF Step(_totalStepNumber - 1, TRUE, CONCAT('Step ', INT_TO_STRING(_totalStepNumber - 1))) THEN
        CompleteSequence();
    END_IF
END_IF

IF _sequenceRun = 6 OR _sequenceRun = 8 OR _sequenceRun = 9 THEN
    _StepBackward();

    IF Step(0, TRUE, 'Step 0') THEN
        StepCompleteWhen(TRUE);
    END_IF

    FOR i := 1 TO _totalStepNumber - 2 DO
        Step(i, TRUE, CONCAT('Step ', INT_TO_STRING(i)));
    END_FOR

    IF Step(_totalStepNumber-1, TRUE, CONCAT('Step ', INT_TO_STRING(_totalStepNumber-1))) THEN
        CompleteSequence();
    END_IF
END_IF

IF _sequenceRun = 7 THEN
    RequestStep(1);

    IF Step(0, TRUE, 'Step 0') THEN
        StepCompleteWhen(TRUE);
    END_IF

    FOR i := 1 TO _totalStepNumber - 2 DO
        Step(i, TRUE, CONCAT('Step ', INT_TO_STRING(i)));
    END_FOR

    IF Step(_totalStepNumber-1, TRUE, CONCAT('Step ', INT_TO_STRING(_totalStepNumber-1))) THEN
        CompleteSequence();
    END_IF
END_IF
END_METHOD

METHOD MAIN_StepModeStepForwardFromRunningStep 
VAR 
	i : INT;
END_VAR
IF _sequenceRun = 1 THEN
    _StepIn();
END_IF

IF _sequenceRun = 11 THEN
    _StepForward();
END_IF

Step(0, TRUE, 'Step 0');
Step(1, TRUE, 'Step 1');

IF Step(2, TRUE, 'Step 2') THEN
    _StepCompleteWhen(_sequenceRun >= 20);
END_IF

IF Step(3, TRUE, 'Step 3') THEN
    _StepCompleteWhen(_sequenceRun >= 20);
END_IF

FOR i := 4 TO _totalStepNumber - 2 DO
    Step(i, TRUE, CONCAT('Step ', INT_TO_STRING(i)));
END_FOR

IF Step(_totalStepNumber-1, TRUE, CONCAT('Step ', INT_TO_STRING(_totalStepNumber-1))) THEN
    CompleteSequence();
END_IF
END_METHOD

METHOD MAIN_StepModeStepIn 
VAR 
	i : INT;
END_VAR
IF _sequenceRun = 1 THEN
    IF Step(0, TRUE, 'Initial step') THEN
        StepCompleteWhen(TRUE);
    END_IF

    FOR i := 1 TO _totalStepNumber - 2 DO
        Step(i, TRUE, CONCAT('Step ', INT_TO_STRING(i)));
    END_FOR

    IF Step(_totalStepNumber-1, TRUE, CONCAT('Step ', INT_TO_STRING(_totalStepNumber-1))) THEN
        _SequenceComplete();
    END_IF
END_IF

IF _sequenceRun > 1 THEN
    IF _currentStep.Status = 20 THEN
       _StepIn();
    END_IF

    // Step 0
    IF Step(0, TRUE, 'Step 0') THEN
        StepCompleteWhen(TRUE);
    END_IF

    // Step 1
    IF Step(1, TRUE, 'Step 1') THEN
        StepCompleteWhen(TRUE);
    END_IF

    // Step 2
    IF Step(2, TRUE, 'Step 2') THEN
        StepCompleteWhen(TRUE);
    END_IF

    // Step 3
    IF Step(3, TRUE, 'Step 3') THEN
        StepCompleteWhen(FALSE);
    END_IF

    FOR i := 4 TO _totalStepNumber - 2 DO
        Step(i, TRUE, CONCAT('Step  ', INT_TO_STRING(i)));
    END_FOR

    IF Step(_totalStepNumber-1, TRUE, CONCAT('Step  ', INT_TO_STRING(_totalStepNumber-1))) THEN
        _SequenceComplete();
    END_IF
END_IF
END_METHOD

METHOD MAIN_StepModeStepInDetailed 
VAR 
	i : INT;
END_VAR
IF _sequenceRun = 1 OR _sequenceRun = 5 THEN
    FOR i := 0 TO _totalStepNumber - 2 DO
        Step(i, TRUE, CONCAT('Step ', INT_TO_STRING(i)));
    END_FOR

    IF Step(_totalStepNumber - 1, TRUE, CONCAT('Step ', INT_TO_STRING(_totalStepNumber - 1))) THEN
        CompleteSequence();
    END_IF
END_IF

IF _sequenceRun = 2 THEN
    _StepIn();

    IF Step(0, TRUE, 'Step 0') THEN
        StepCompleteWhen(TRUE);
    END_IF

    FOR i := 1 TO _totalStepNumber - 2 DO
        Step(i, TRUE, CONCAT('Step ', INT_TO_STRING(i)));
    END_FOR

    IF Step(_totalStepNumber - 1, TRUE, CONCAT('Step ', INT_TO_STRING(_totalStepNumber - 1))) THEN
        CompleteSequence();
    END_IF
END_IF

IF _sequenceRun = 3 OR _sequenceRun = 4 THEN
    _StepIn();

    IF Step(0, TRUE, 'Step 0') THEN
        StepCompleteWhen(TRUE);
    END_IF

    IF Step(1, TRUE, 'Step 1') THEN
        RequestStep(_totalStepNumber - 1);
    END_IF

    FOR i := 2 TO _totalStepNumber - 2 DO
        Step(i, TRUE, CONCAT('Step ', INT_TO_STRING(i)));
    END_FOR

    IF Step(_totalStepNumber - 1, TRUE, CONCAT('Step ', INT_TO_STRING(_totalStepNumber - 1))) THEN
        CompleteSequence();
    END_IF
END_IF
END_METHOD

METHOD MAIN_StepModeUncommentPartOfRunningSequencer 
VAR 
	i : INT;
END_VAR
IF _sequenceRun = 1 THEN
    IF (_currentStep.Status = 20) THEN
        _StepIn();
    END_IF

    IF Step(0, TRUE, 'Step 0') THEN
        StepCompleteWhen(TRUE);
    END_IF

    //	IF Step(1, TRUE, 'Step 1') THEN
    //	   StepCompleteWhen(TRUE);
    //	END_IF
    //	IF Step(2, TRUE, 'Step 2') THEN
    //	   StepCompleteWhen(TRUE);
    //	END_IF
    IF Step(3, TRUE, 'Step 3') THEN
        StepCompleteWhen(FALSE);
    END_IF

    FOR i := 4 TO _totalStepNumber - 2 DO
        IF Step(i, TRUE, CONCAT('Step ', INT_TO_STRING(i))) THEN
            StepCompleteWhen(FALSE);
        END_IF
    END_FOR

    IF Step(_totalStepNumber-1, TRUE, CONCAT('Step ', INT_TO_STRING(_totalStepNumber-1))) THEN
        _SequenceComplete();
    END_IF
END_IF

IF _sequenceRun = 2 THEN
    IF (_currentStep.Status = 20) THEN
        _StepIn();
    END_IF

    IF Step(0, TRUE, 'Step 0') THEN
        StepCompleteWhen(TRUE);
    END_IF

    IF Step(1, TRUE, 'Step 1') THEN
        StepCompleteWhen(TRUE);
    END_IF

    IF Step(2, TRUE, 'Step 2') THEN
        StepCompleteWhen(TRUE);
    END_IF

    IF Step(3, TRUE, 'Step 3') THEN
        StepCompleteWhen(FALSE);
    END_IF

    FOR i := 4 TO _totalStepNumber - 2 DO
        IF Step(i, TRUE, CONCAT('Step ', INT_TO_STRING(i))) THEN
            StepCompleteWhen(FALSE);
        END_IF
    END_FOR

    IF Step(_totalStepNumber-1, TRUE, CONCAT('Step ', INT_TO_STRING(_totalStepNumber-1))) THEN
        _SequenceComplete();
    END_IF
END_IF
END_METHOD

METHOD MAIN_SwitchStepModeOnDuringStepExecution 
VAR 
	i : INT;
END_VAR
IF _sequenceRun = 1 THEN
    IF Step(0, TRUE, 'Step 0') THEN
        StepCompleteWhen(TRUE);
    END_IF

    IF Step(1, TRUE, 'Step 1') THEN
        StepCompleteWhen(FALSE);
    END_IF

    FOR i := 2 TO _totalStepNumber - 2 DO
        Step(i, TRUE, CONCAT('Step ', INT_TO_STRING(i)));
    END_FOR

    IF Step(_totalStepNumber-1, TRUE, CONCAT('Step ', INT_TO_STRING(_totalStepNumber-1))) THEN
        CompleteSequence();
    END_IF
END_IF

IF _sequenceRun > 1 THEN
    IF Step(0, TRUE, 'Step 0') THEN
        StepCompleteWhen(TRUE);
    END_IF

    IF Step(1, TRUE, 'Step 1') THEN
		IF _sequenceRun >=5 THEN
			SetStepMode();
		END_IF
        StepCompleteWhen(_sequenceRun >=10);
    END_IF

    FOR i := 2 TO _totalStepNumber - 2 DO
        Step(i, TRUE, CONCAT('Step ', INT_TO_STRING(i)));
    END_FOR

    IF Step(_totalStepNumber-1, TRUE, CONCAT('Step ', INT_TO_STRING(_totalStepNumber-1))) THEN
        CompleteSequence();
    END_IF
END_IF
END_METHOD

METHOD MAIN_SwitchStepModeStepOffFromReadyToRun 
VAR 
	i : INT;
END_VAR
SetCyclicMode();
Step(0, TRUE, 'Step 0');
Step(1, TRUE, 'Step 1');

IF Step(2, TRUE, 'Step 2') THEN
    _StepCompleteWhen(_sequenceRun >= 20);
END_IF

IF Step(3, TRUE, 'Step 3') THEN
    _StepCompleteWhen(_sequenceRun >= 20);
END_IF

FOR i := 4 TO _totalStepNumber - 2 DO
    Step(i, TRUE, CONCAT('Step ', INT_TO_STRING(i)));
END_FOR

IF Step(_totalStepNumber-1, TRUE, CONCAT('Step ', INT_TO_STRING(_totalStepNumber-1))) THEN
    CompleteSequence();
END_IF
END_METHOD

METHOD MAIN_SwitchStepModeStepOffFromRunning 
VAR 
	i : INT;
END_VAR
SetCyclicMode();
Step(0, TRUE, 'Step 0');
Step(1, TRUE, 'Step 1');

IF Step(2, TRUE, 'Step 2') THEN
    _StepCompleteWhen(_sequenceRun >= 20);
END_IF

IF Step(3, TRUE, 'Step 3') THEN
    _StepCompleteWhen(_sequenceRun >= 20);
END_IF

FOR i := 4 TO _totalStepNumber - 2 DO
    Step(i, TRUE, CONCAT('Step ', INT_TO_STRING(i)));
END_FOR

IF Step(_totalStepNumber-1, TRUE, CONCAT('Step ', INT_TO_STRING(_totalStepNumber-1))) THEN
    CompleteSequence();
END_IF
END_METHOD

METHOD MAIN_SwitchStepModeStepOnFromRunning 
VAR 
	i : INT;
END_VAR
SetStepMode();
Step(0, TRUE, 'Step 0');
Step(1, TRUE, 'Step 1');

IF Step(2, TRUE, 'Step 2') THEN
    _StepCompleteWhen(_sequenceRun >= 20);
END_IF

IF Step(3, TRUE, 'Step 3') THEN
    _StepCompleteWhen(_sequenceRun >= 20);
END_IF

FOR i := 4 TO _totalStepNumber - 2 DO
    Step(i, TRUE, CONCAT('Step ', INT_TO_STRING(i)));
END_FOR

IF Step(_totalStepNumber-1, TRUE, CONCAT('Step ', INT_TO_STRING(_totalStepNumber-1))) THEN
    CompleteSequence();
END_IF
END_METHOD

METHOD MAIN_UncommentPartOfRunningSequencer 
VAR 
	i : INT;
END_VAR
IF _sequenceRun =1 THEN
	IF Step(0, TRUE, 'Step 0') THEN
	   StepCompleteWhen(TRUE);
	END_IF

//	IF Step(1, TRUE, 'Step 1') THEN
//	   StepCompleteWhen(TRUE);
//	END_IF

//	IF Step(2, TRUE, 'Step 2') THEN
//	   StepCompleteWhen(TRUE);
//	END_IF

	IF Step(3, TRUE, 'Step 3') THEN
	   StepCompleteWhen(FALSE);
	END_IF
	
	FOR i := 4 TO _totalStepNumber-2 DO
		IF Step(i, TRUE, CONCAT('Step ', INT_TO_STRING(i))) THEN
			StepCompleteWhen(FALSE);
		END_IF
	END_FOR
	
	IF Step(_totalStepNumber-1, TRUE, CONCAT('Step ', INT_TO_STRING(_totalStepNumber-1))) THEN
	  _SequenceComplete();
	END_IF
END_IF

IF _sequenceRun =2 THEN
	IF Step(0, TRUE, 'Step 0') THEN
	   StepCompleteWhen(TRUE);
	END_IF

	IF Step(1, TRUE, 'Step 1') THEN
	   StepCompleteWhen(TRUE);
	END_IF

	IF Step(2, TRUE, 'Step 2') THEN
	   StepCompleteWhen(TRUE);
	END_IF

	IF Step(3, TRUE, 'Step 3') THEN
			StepCompleteWhen(FALSE);
	END_IF
	
	FOR i := 4 TO _totalStepNumber-2 DO
		IF Step(i, TRUE, CONCAT('Step ', INT_TO_STRING(i))) THEN
			StepCompleteWhen(FALSE);
		END_IF
	END_FOR
	
	IF Step(_totalStepNumber-1, TRUE, CONCAT('Step ', INT_TO_STRING(_totalStepNumber-1))) THEN
	  _SequenceComplete();
	END_IF
END_IF
END_METHOD

METHOD PROTECTED OnRestore
_restoreCycleCount := _restoreCycleCount + 1;
END_METHOD

METHOD PROTECTED OnSequenceCompleted
_onSequenceCompleteCount := _onSequenceCompleteCount + 1;
END_METHOD

METHOD PROTECTED OnSequencerError
VAR_INPUT
	inErrorId : eSequencerError;
END_VAR
CASE inErrorId OF
	eSequencerError.noError :
		_onSequencerErrorCount := _onSequencerErrorCount + 0;
	eSequencerError.NotUniqueStepId :
		_onSequencerErrorCount := _onSequencerErrorCount + 10;
	eSequencerError.StepIdHasBeenChanged :
		_onSequencerErrorCount := _onSequencerErrorCount + 20;
	eSequencerError.OrderOfTheStepHasBeenChanged :
		_onSequencerErrorCount := _onSequencerErrorCount + 40;
	eSequencerError.StepWithRequestedIdDoesNotExists :
		_onSequencerErrorCount := _onSequencerErrorCount + 50;
	eSequencerError.MultipleRequestStepMethodCall :
		_onSequencerErrorCount := _onSequencerErrorCount + 60;
	eSequencerError.StepIdTooLow :
		_onSequencerErrorCount := _onSequencerErrorCount + 70;
	eSequencerError.StepIdTooHigh :
		_onSequencerErrorCount := _onSequencerErrorCount + 80;
	ELSE
		_onSequencerErrorCount := _onSequencerErrorCount + 0;
END_CASE
END_METHOD

METHOD PROTECTED OnStateChange
VAR_INPUT
	PreviousState	: INT;
	NewState 		: INT;
END_VAR
THIS^._onStateChangeCount := THIS^._onStateChangeCount + 1;

_stateChangeFrom := PreviousState;
_stateChangeTo := NewState;

IF _callRestoreInOnStateChange THEN
	Restore();
END_IF
END_METHOD

METHOD PROTECTED OnStepCompleted
_onCompleteStepCount := _onCompleteStepCount + 1;
END_METHOD

PROPERTY PostOpenRequestStepCycle : UINT
GET
PostOpenRequestStepCycle := _postOpenRequestStepCycle;
END_GET
SET
_postOpenRequestStepCycle := PostOpenRequestStepCycle;
END_SET
END_PROPERTY

PROPERTY PreCloseRequestStepCycle : UINT
GET
PreCloseRequestStepCycle := _preCloseRequestStepCycle;
END_GET
SET
_preCloseRequestStepCycle := PreCloseRequestStepCycle;
END_SET
END_PROPERTY

PROPERTY ReqStep : INT
GET
ReqStep := _reqStep;
END_GET
SET
_reqStep := ReqStep;
END_SET
END_PROPERTY

PROPERTY ReqStepNotExists : INT
GET
ReqStepNotExists := _reqStepNotExists;
END_GET
SET
_reqStepNotExists:=ReqStepNotExists;
END_SET
END_PROPERTY

PROPERTY INTERNAL RequestStepCycle : UINT
GET
RequestStepCycle := _requestStepCycle;
END_GET
SET
_requestStepCycle := RequestStepCycle;
END_SET
END_PROPERTY

PROPERTY RunAllSteps : BOOL
GET
RunAllSteps := _runAllSteps;
END_GET
SET
_runAllSteps := RunAllSteps;
END_SET
END_PROPERTY

PROPERTY RunOneStep : BOOL
GET
RunOneStep := _runOneStep;
END_GET
SET
_runOneStep := RunOneStep;
END_SET
END_PROPERTY

{attribute 'TcRpcEnable'}
METHOD SaveNumberOfStepsInSequence
_numberOfSteps := THIS^._numberOfStepsInSequence;
_previousNumberOfSteps	:= THIS^._previousNumberOfStepsInSequence;
END_METHOD

PROPERTY SequenceCycles : UINT
GET
SequenceCycles := _sequenceCycles;
END_GET
SET
_sequenceCycles := SequenceCycles;
END_SET
END_PROPERTY

METHOD INTERNAL SequencerClose
SUPER^._Close();
END_METHOD

METHOD INTERNAL SequencerOpen
SUPER^._Open();
END_METHOD

PROPERTY SequenceRun : ULINT
GET
SequenceRun := _sequenceRun;
END_GET
SET
_sequenceRun:=SequenceRun;
END_SET
END_PROPERTY

{attribute 'TcRpcEnable'}
METHOD INTERNAL SetChildState 
VAR_INPUT
	inState			:	INT;
END_VAR
THIS^._myTcoChildState.ChangeState(inState);
END_METHOD

{attribute 'TcRpcEnable'}
METHOD INTERNAL SetCurrentStep 
VAR_INPUT
	inStepID 			:	INT;
	inStepDescription	:	STRING(254);
END_VAR
THIS^._currentStep.ID			:=	inStepID;
THIS^._currentStep.Description	:=	inStepDescription;
END_METHOD

{attribute 'TcRpcEnable'}
METHOD SetCurrentStepToErrorState : BOOL
_currentStep.Status := TcoCore.eStepStatus.Error;

SetCurrentStepToErrorState := _currentStep.Status = TcoCore.eStepStatus.Error;
END_METHOD

METHOD SetCyclicMode : BOOL
ModeController.Mode := eSequencerMode.CyclicMode;

SetCyclicMode := ModeController.Mode = eSequencerMode.CyclicMode;
END_METHOD

{attribute 'TcRpcEnable'}
METHOD SetInvalidMode : BOOL
ModeController.Mode := eSequencerMode.Invalid;

SetInvalidMode := ModeController.Mode = eSequencerMode.Invalid;
END_METHOD

METHOD INTERNAL SetNumberOfSteps 
VAR_INPUT
	inNumberOfSteps : UINT;
END_VAR
_stepCounter 						:=	inNumberOfSteps;
_numberOfStepsInSequence			:=	inNumberOfSteps;
_previousNumberOfStepsInSequence 	:=	inNumberOfSteps;
END_METHOD

METHOD INTERNAL SetSequenceAsChecked
_stepIDUniquenessChecked := TRUE;
_StepIdUniquenessControlState := eStepIdUniquenessControlState.Done;
END_METHOD

METHOD INTERNAL SetSequenceAsNotChecked
_stepIDUniquenessChecked := FALSE;
_StepIdUniquenessControlState := eStepIdUniquenessControlState.NotYetStarted;
END_METHOD

METHOD SetStepMode : BOOL
ModeController.Mode := eSequencerMode.StepMode;

SetStepMode := ModeController.Mode = eSequencerMode.StepMode;
END_METHOD

{attribute 'TcRpcEnable'}
METHOD INTERNAL SetupChildRequestedState 
VAR_INPUT
	inState			:	INT;
END_VAR
THIS^._myTcoChildState.RequestedState:=inState;
END_METHOD

PROPERTY StepDescription : STRING(254);
GET
StepDescription := _stepDescription;
END_GET
SET
_stepDescription := StepDescription;
END_SET
END_PROPERTY

PROPERTY StepId : INT
GET
StepId := _stepId;
END_GET
SET
_stepId := StepId;
END_SET
END_PROPERTY

PROPERTY StepInEvents : UINT
GET
StepInEvents := _stepInEvents;
END_GET
SET
_stepInEvents := StepInEvents;
END_SET
END_PROPERTY

PROPERTY TcoSequencerTest : eTcoSequencerTests
GET
TcoSequencerTest := _tcoSequencerTest;
END_GET
SET
_tcoSequencerTest := TcoSequencerTest;
END_SET
END_PROPERTY

PROPERTY TotalStepNumber : UINT
GET
TotalStepNumber := _totalStepNumber;
END_GET
SET
_totalStepNumber := TotalStepNumber;
END_SET
END_PROPERTY

END_FUNCTION_BLOCK

(* stored: Version 1.1.0.1
   POU TcoSequencerTestType: Id {fcbfa856-fa22-0d81-1570-4e6ea8af1a6a}, SpecialFunc None
   Folder _Tests: Id {da5f6f87-5f5f-0a79-3f5a-77ea7614efba}
   Folder MAINS: Id {acde229d-7801-0426-1307-56c91d523529}
   Method _RequestStep: Id {c341729a-ee0f-0c81-387e-76f75b84ca5c}
   Method _SequenceComplete: Id {85f5b06a-adec-0445-17bd-b4a5a342dd3f}
   Method _Step: Id {fe082966-d27d-07ef-1434-1d037dbf0efd}
   Method _StepBackward: Id {5f585814-394a-08f9-0771-c464e15549a9}
   Method _StepCompleteWhen: Id {ecbc01f9-58db-026e-1bf5-c5846075a6fe}
   Method _StepForward: Id {1336721c-30ea-0034-17f3-d59f4eee23cd}
   Method _StepIn: Id {ee94a64e-dfb7-0a77-170b-40a3b6ed768d}
   Property CallRestoreInOnStateChange: Id {e4bdc12d-4c4a-05b0-2eef-3193c2915dfb}
   Get Get: Id {da157f44-3b5f-0e32-3222-e45b28409abf}
   Set Set: Id {4dd8aef3-f2f1-0f9b-2672-9322f8705c35}
   Method ChildHasAutoRestoreEnabled: Id {d10b079a-4f99-0c33-1169-fdd0ae5abb4a}
   Method ChildIsAutoRestorable: Id {6a713271-9048-0703-3c9a-9780e01c1ba9}
   Method ClearNumberOfSteps: Id {53185e96-25c2-084b-37ed-a715d9a18864}
   Property CyclicCycles: Id {bafb42e5-b1cc-0784-30ac-cfeef85702f9}
   Get Get: Id {debb9782-9b85-070b-1cb6-b2014e29c9e5}
   Set Set: Id {b924469d-2ea2-0632-0149-336ec4e42fbc}
   Property Enabled: Id {3b6a30b8-3bf9-0527-1061-ff7665615f52}
   Get Get: Id {7340ea50-4fe8-063b-205b-ebd3fc87915a}
   Set Set: Id {c443b63f-06ef-00d9-1acc-f8408ef8de77}
   Property FinishStep: Id {dbdca6ba-1654-0ccb-110e-5039e44fd003}
   Get Get: Id {75c52477-2552-0c90-3c28-c4f495fc1b9e}
   Set Set: Id {854ed8a2-1462-0d2c-0ded-bccf07b449fb}
   Method GetChildState: Id {c16345a9-5d5f-0dd8-1791-5222c9847257}
   Method GetOrderOfTheCurrentlyEvaluatedStep: Id {64b5d6a9-df51-0a21-3b1f-b671ca6be73d}
   Method GetOrderOfTheCurrentlyExecutedStep: Id {902a04f9-38ed-088d-1f52-ba3e349f4809}
   Method GetRequestStepCycle: Id {4d5a7304-be22-0f43-1824-10365a464aee}
   Method HasAutoRestoreEnabled: Id {2f7d97be-7276-0c05-2a6b-80bd3ac53780}
   Property InitReqStepCycle: Id {ba0afa3b-02d8-05b1-1f94-cb4cb35070ef}
   Get Get: Id {b2c3c996-b02d-0932-011c-b734f124c551}
   Set Set: Id {4ad57638-577d-035c-09c8-87bea651c375}
   Method IsAutoRestorable: Id {755204b0-6ac7-0749-0ee2-4831cf006a59}
   Method Main: Id {c539ed7e-eed2-0192-1223-93740507fed3}
   Method MAIN_ChangeStepIdDuringExecution: Id {7325dc63-03fc-0cb6-3905-c7f8d095eb41}
   Method MAIN_CheckStepIdUniqueness: Id {15a3e7dc-74f2-02a3-2ac1-d30e7a4012ce}
   Method MAIN_CommentOutPartOfRunningSequencer: Id {cdc055fb-5045-0554-359e-f41e9edc10d0}
   Method MAIN_ExecutionInOnePLCcycle: Id {82bf9e1e-488e-052a-10d3-9785fac50ab5}
   Method MAIN_MaxStepId: Id {89c57b91-7969-0bc0-1dba-e185486115a0}
   Method MAIN_MinStepId: Id {3db71dd8-2beb-09ca-0629-9aa5ac8685f7}
   Method MAIN_NumberOfStepsCount: Id {b05ad8eb-06f5-0cda-2076-ec8cf7a4be79}
   Method MAIN_OnStateChangeWhenChangingModes: Id {5523946f-df40-0fd4-33fa-fc8da62df1a4}
   Method MAIN_RequestStep: Id {4c0d54af-8ae2-071b-3a28-1389f6d935e6}
   Method MAIN_RequestStepFromHigherToLower: Id {419bf385-41fb-036e-3170-06e9de257e55}
   Method MAIN_RequestStepFromLowerToHigher: Id {c9a7c0f6-3cd8-06c0-0301-9fe1b94f02d6}
   Method MAIN_RequestStepToFirstStepWithStepId0: Id {6a25be65-f058-0e20-0e3b-937bad0f5ca9}
   Method MAIN_RequestStepToNotExistingStep: Id {ab1f2097-baf0-0820-0fa7-f7d70b1b885a}
   Method MAIN_RequestStepWhilePreviousRequestStepHasNotBeenYetProcessed: Id {28dfbafc-2ae7-031e-22ce-2f4a5142d5d3}
   Method MAIN_RestoreChildBetweenSteps: Id {ac2289b4-bd06-01af-3bac-dde62540b496}
   Method MAIN_SetStepMode: Id {d576efc9-c913-07c2-0f81-b007e9cd1adf}
   Method MAIN_StepMode: Id {1ec61e0e-5a4e-0084-3582-dae83fa6fec5}
   Method MAIN_StepModeChangeStepIdDuringExecution: Id {74bb999f-bcf5-00d2-09c0-221d08724c79}
   Method MAIN_StepModeChangeStepOrder: Id {a18e7779-2fd1-0217-19f5-e66cf5666c91}
   Method MAIN_StepModeCommentOutPartOfRunningSequencer: Id {aaab85d5-8141-0ebd-27c0-46f7c13e56d4}
   Method MAIN_StepModeDisabledStep: Id {5fe3466f-6208-065a-1099-5c8f566b4fab}
   Method MAIN_StepModeRequestStepFromHigherToLower: Id {305ecba4-6af4-0c13-0243-4db4c133c944}
   Method MAIN_StepModeRequestStepFromLowerToHigher: Id {fccb1663-b375-08d8-129e-f3ab0bf97615}
   Method MAIN_StepModeStepBackwardFromRunningStep: Id {812332ac-f7f0-0ad6-2f79-dc3c3570d1be}
   Method MAIN_StepModeStepForwardBackward: Id {f96ebcfa-a209-020c-2e79-9c9472e48b8b}
   Method MAIN_StepModeStepForwardFromRunningStep: Id {8811e73c-bd43-05be-112e-c4273e1ea192}
   Method MAIN_StepModeStepIn: Id {0390dd02-1a10-0073-1e38-93414f7de3c0}
   Method MAIN_StepModeStepInDetailed: Id {caafe3d1-a672-09d8-3231-17110072d530}
   Method MAIN_StepModeUncommentPartOfRunningSequencer: Id {9fbb406b-f64b-09a7-0a13-18757c50d2de}
   Method MAIN_SwitchStepModeOnDuringStepExecution: Id {82a07c31-d734-0f81-22b3-4e8a8e886550}
   Method MAIN_SwitchStepModeStepOffFromReadyToRun: Id {4a5fa1c4-6a93-0a96-21f0-c372d23fecef}
   Method MAIN_SwitchStepModeStepOffFromRunning: Id {b12b71a8-cd05-0127-2425-292580190aa7}
   Method MAIN_SwitchStepModeStepOnFromRunning: Id {4f7b667c-e463-019e-1471-cf271e293caa}
   Method MAIN_UncommentPartOfRunningSequencer: Id {a9013512-a01a-0b7c-0e2d-57715e51a07d}
   Method OnRestore: Id {a9b6abd9-864a-0bb5-33cb-25bef86aee6c}
   Method OnSequenceCompleted: Id {4225e218-d628-0ae3-358d-91569294365a}
   Method OnSequencerError: Id {b05bb29d-c819-0dda-10d0-2c6364c65570}
   Method OnStateChange: Id {abdcb0ab-194d-0554-2b0b-52924360c478}
   Method OnStepCompleted: Id {3a298859-30d7-0987-2b70-6199d376e9e5}
   Property PostOpenRequestStepCycle: Id {7b8f04ee-820a-0719-0199-bb6e9089b7df}
   Get Get: Id {a321aee8-8b16-0f83-189f-821d34d2e961}
   Set Set: Id {febb691e-5ae2-0c85-20f7-b608221c5a6a}
   Property PreCloseRequestStepCycle: Id {f57d8156-cb77-0043-2d3a-081ce498e6b3}
   Get Get: Id {60745cad-3d46-07d2-3e05-44bb7167dcb9}
   Set Set: Id {df019169-25c9-08a2-2622-abc5bd2dba53}
   Property ReqStep: Id {78240d3c-e450-0617-3646-a8723c629e53}
   Get Get: Id {c1898996-4e34-083b-327b-4f6e9a318ff3}
   Set Set: Id {d8e5dcd7-3bd8-01a2-0742-6d134f7e9c8f}
   Property ReqStepNotExists: Id {55e8c9ed-9c7a-0420-17ff-b372c640515c}
   Get Get: Id {a9473ac0-47ad-0df9-2d18-893379b0397e}
   Set Set: Id {d0246ddc-2383-08f9-3a2c-db14be630c48}
   Property RequestStepCycle: Id {d445b6db-77f8-05eb-0ee7-ef5085c25b2d}
   Get Get: Id {430b2ff2-9b2c-089e-158b-a3d2549ef774}
   Set Set: Id {ecc154d3-1884-0521-172a-f144fedd707e}
   Property RunAllSteps: Id {2581a28d-9821-076f-0c4e-25e91de855b1}
   Get Get: Id {e96c518e-08c2-01ad-133d-5734d5b50540}
   Set Set: Id {2a61b193-7b88-0d6f-1e80-9c1d1245fc0d}
   Property RunOneStep: Id {647d1f4c-c801-0a7d-3637-03fad2763e6a}
   Get Get: Id {0a227db8-c6b6-046a-2249-e7f145fb9881}
   Set Set: Id {6db3a246-4857-01e3-1276-b995832ca587}
   Method SaveNumberOfStepsInSequence: Id {5db122d9-3e40-0829-2aab-06d2c5882841}
   Property SequenceCycles: Id {98b89647-dd89-049d-3935-41d364281ed5}
   Get Get: Id {626a3d78-1d84-0cbf-370f-36babee53df1}
   Set Set: Id {49396dde-5339-04f0-004d-dd714d9d96d8}
   Method SequencerClose: Id {c7506de2-f987-0a3e-1e2e-7d504bcf9174}
   Method SequencerOpen: Id {17f85c5f-06f4-018f-28b3-f696a56ed990}
   Property SequenceRun: Id {cd544d0d-0747-0358-2ad8-13e2cea5f814}
   Get Get: Id {4e19fad3-dc68-0179-30cc-b90b005e0e52}
   Set Set: Id {8ad874a4-06ab-0b53-015c-5054e178e3a2}
   Method SetChildState: Id {7ba9f2cb-a634-0387-3c1a-0f23e9f68d57}
   Method SetCurrentStep: Id {c2e081c2-228a-0888-0a3e-167c8f2e5624}
   Method SetCurrentStepToErrorState: Id {a977cb4b-07ef-02fa-0488-3b603d70a523}
   Method SetCyclicMode: Id {46dddda7-6cc4-09bf-260a-7edfd4351354}
   Method SetInvalidMode: Id {fb68baca-d798-08d1-1d73-8980db47120d}
   Method SetNumberOfSteps: Id {12dd8dee-1aee-0992-3de9-66e4ddfe479e}
   Method SetSequenceAsChecked: Id {3100e91a-0746-0506-3138-6c4b89b39740}
   Method SetSequenceAsNotChecked: Id {4f847581-3b2b-010a-27ba-798029208963}
   Method SetStepMode: Id {76cbfb8d-0c45-0ccb-352d-3090bd4ad755}
   Method SetupChildRequestedState: Id {8dd64da9-588e-0694-0dd3-d72dd065b20c}
   Property StepDescription: Id {fc692f65-5380-0ce1-0f50-f3bd5b17b686}
   Get Get: Id {344e5c58-353d-0aa7-2888-88d944dea49e}
   Set Set: Id {0bba76c1-42ae-0d4e-140c-07a966acc02e}
   Property StepId: Id {3c2d860f-565a-0fa1-32c9-dbda09f6bc7e}
   Get Get: Id {83c9d1f5-77ae-00b9-0e05-56b4a5a96679}
   Set Set: Id {c4236a24-e6ba-01d0-091a-63baa3be093c}
   Property StepInEvents: Id {15993880-527f-0b94-163a-f65c74b3ec10}
   Get Get: Id {f367c089-7bea-0ccc-3e80-91a702cf62ab}
   Set Set: Id {1b50b619-f334-069a-29a2-17c9947ce924}
   Property TcoSequencerTest: Id {fe6d888f-2ebc-04dc-1261-8605c27c5c74}
   Get Get: Id {41e185db-12c1-07ab-0f58-766b5f339b9f}
   Set Set: Id {8d825be0-af7c-0c3f-227d-52ff06c6aa6a}
   Property TotalStepNumber: Id {db2c4ccc-fc3b-021f-02a3-993759add6e0}
   Get Get: Id {bbb16e4d-67b3-0829-1c39-243ecdf53e36}
   Set Set: Id {e1822b47-7b45-0c45-1c60-967714dfb1cb} *)
